(* Logix 5000 project; controller reports 1756-L63 rev 20.15; software revision 20.04; part 43 of 52 *)

        [112].log_data[48].valid := 1, [112].log_data[49].min := 6.5370584, [112].log_data[49].max := 9.345203, [112].log_data[49].total := 30173.871, [112].log_data[49].time := 3600.0, [112].log_data[49].minminute := 59, [112].log_data[49].maxminute := 34, [112].log_data[49].valid := 1, [112].log_data[50].min := 1.828552, [112].log_data[50].max := 1.9386716, [112].log_data[50].total := 6771.5327, [112].log_data[50].time := 3600.0, [112].log_data[50].minminute := 33, [112].log_data[50].maxminute := 40, [112].log_data[50].valid := 1, [112].log_data[51].time := 3600.0, [112].log_data[51].valid := 1, [112].log_data[52].min := -2.7799988, [112].log_data[52].max := 0.11999512, [112].log_data[52].total := -7734.9287, [112].log_data[52].time := 3600.0, [112].log_data[52].minminute := 1, [112].log_data[52].valid := 1, [112].log_data[53].min := -2.7000046, [112].log_data[53].max := 0.13999939, [112].log_data[53].total := -7364.768, [112].log_data[53].time := 3600.0, [112].log_data[53].minminute := 38, [112].log_data[53].maxminute := 27, [112].log_data[53].valid := 1, [112].log_data[54].max := 0.537, [112].log_data[54].total := 1216.9052, [112].log_data[54].time := 3600.0, [112].log_data[54].maxminute := 12, [112].log_data[54].valid := 1, [112].log_data[55].max := 0.528, [112].log_data[55].total := 1217.3307, [112].log_data[55].time := 3600.0, [112].log_data[55].minminute := 5, [112].log_data[55].maxminute := 38, [112].log_data[55].valid := 1, [112].log_data[56].min := 0.15938194, [112].log_data[56].max := 0.15989229, [112].log_data[56].total := 574.438, [112].log_data[56].time := 3600.0, [112].log_data[56].minminute := 2, [112].log_data[56].maxminute := 17, [112].log_data[56].valid := 1, [112].log_data[57].min := 0.22258775, [112].log_data[57].max := 0.22325513, [112].log_data[57].total := 802.80646, [112].log_data[57].time := 3600.0, [112].log_data[57].minminute := 59, [112].log_data[57].maxminute := 9, [112].log_data[57].valid := 1, [112].log_data[58].time := 3600.0, [112].log_data[58].valid := 1, [112].log_data[59].time := 3600.0, [112].log_data[59].valid := 1, [112].log_data[60].valid := 1,
        [112].log_data[61].valid := 1, [112].log_data[62].valid := 1, [112].log_data[63].valid := 1, [112].log_data[64].valid := 1, [112].log_data[65].valid := 1, [112].log_data[66].valid := 1, [112].log_data[67].valid := 1, [112].log_data[68].valid := 1, [112].log_data[69].valid := 1, [112].log_data[70].valid := 1, [112].log_data[71].valid := 1, [112].log_data[72].valid := 1, [112].log_data[73].valid := 1, [112].log_data[74].valid := 1, [112].log_data[75].valid := 1, [112].log_data[76].valid := 1, [112].log_data[77].valid := 1, [112].log_data[78].valid := 1, [112].log_data[79].valid := 1, [112].log_data[80].valid := 1, [112].log_data[81].valid := 1, [112].log_data[82].valid := 1, [112].log_data[83].valid := 1, [112].log_data[84].valid := 1, [112].log_data[85].valid := 1, [112].log_data[86].valid := 1, [112].log_data[87].valid := 1, [112].log_data[88].valid := 1, [112].log_data[89].valid := 1, [112].log_data[90].valid := 1, [112].log_data[91].valid := 1, [112].log_data[92].valid := 1, [112].log_data[93].valid := 1, [112].log_data[94].valid := 1, [112].log_data[95].valid := 1, [112].log_data[96].valid := 1, [112].log_data[97].valid := 1, [112].log_data[98].valid := 1, [112].log_data[99].valid := 1, [112].log_data[100].valid := 1, [112].log_data[101].valid := 1, [112].log_data[102].valid := 1, [112].log_data[103].valid := 1, [112].log_data[104].valid := 1, [112].log_data[105].valid := 1, [112].log_data[106].valid := 1, [112].log_data[107].valid := 1, [112].log_data[108].valid := 1, [112].log_data[109].valid := 1, [112].log_data[110].valid := 1, [112].log_data[111].valid := 1, [112].log_data[112].valid := 1, [112].log_data[113].valid := 1, [112].log_data[114].valid := 1, [112].log_data[115].valid := 1, [112].log_data[116].valid := 1, [112].log_data[117].valid := 1, [112].log_data[118].valid := 1, [112].log_data[119].valid := 1, [112].log_data[120].valid := 1,
        [112].log_data[121].valid := 1, [112].log_data[122].valid := 1, [112].log_data[123].valid := 1, [112].log_data[124].valid := 1, [112].time.Year := 2023, [112].time.Month := 1, [112].time.Day := 17, [112].time.Hour := 19, [112].time.Minute := 59, [112].time.Second := 59, [113].log_data[0].min := 1.0, [113].log_data[0].max := 1.0, [113].log_data[0].total := 3599.5, [113].log_data[0].time := 3599.5, [113].log_data[0].valid := 1, [113].log_data[1].max := 1.0, [113].log_data[1].total := 584.0, [113].log_data[1].time := 3599.5, [113].log_data[1].maxminute := 41, [113].log_data[1].valid := 1, [113].log_data[2].max := 1.0, [113].log_data[2].total := 580.5, [113].log_data[2].time := 3599.5, [113].log_data[2].maxminute := 41, [113].log_data[2].valid := 1, [113].log_data[3].time := 3599.5, [113].log_data[3].valid := 1, [113].log_data[4].time := 3599.5, [113].log_data[4].valid := 1, [113].log_data[5].max := 1.0, [113].log_data[5].total := 240.0, [113].log_data[5].time := 3599.5, [113].log_data[5].maxminute := 44, [113].log_data[5].valid := 1, [113].log_data[6].time := 3599.5, [113].log_data[6].valid := 1, [113].log_data[7].time := 3599.5, [113].log_data[7].valid := 1, [113].log_data[8].min := 1.0, [113].log_data[8].max := 1.0, [113].log_data[8].total := 3599.5, [113].log_data[8].time := 3599.5, [113].log_data[8].valid := 1, [113].log_data[9].min := 1.0, [113].log_data[9].max := 1.0, [113].log_data[9].total := 3599.5, [113].log_data[9].time := 3599.5, [113].log_data[9].valid := 1, [113].log_data[10].min := 1.0, [113].log_data[10].max := 1.0, [113].log_data[10].total := 3599.5, [113].log_data[10].time := 3599.5, [113].log_data[10].valid := 1, [113].log_data[11].time := 3599.5, [113].log_data[11].valid := 1, [113].log_data[12].min := 1.0, [113].log_data[12].max := 1.0, [113].log_data[12].total := 3599.5, [113].log_data[12].time := 3599.5, [113].log_data[12].valid := 1,
        [113].log_data[13].min := 1.0, [113].log_data[13].max := 1.0, [113].log_data[13].total := 3599.5, [113].log_data[13].time := 3599.5, [113].log_data[13].valid := 1, [113].log_data[14].time := 3599.5, [113].log_data[14].valid := 1, [113].log_data[15].time := 3599.5, [113].log_data[15].valid := 1, [113].log_data[16].time := 3599.5, [113].log_data[16].valid := 1, [113].log_data[17].min := 1.0, [113].log_data[17].max := 1.0, [113].log_data[17].total := 3599.5, [113].log_data[17].time := 3599.5, [113].log_data[17].valid := 1, [113].log_data[18].time := 3599.5, [113].log_data[18].valid := 1, [113].log_data[19].time := 3599.5, [113].log_data[19].valid := 1, [113].log_data[20].time := 3599.5, [113].log_data[20].valid := 1, [113].log_data[21].min := 1.0, [113].log_data[21].max := 1.0, [113].log_data[21].total := 3599.5, [113].log_data[21].time := 3599.5, [113].log_data[21].valid := 1, [113].log_data[22].time := 3599.5, [113].log_data[22].valid := 1, [113].log_data[23].time := 3599.5, [113].log_data[23].valid := 1, [113].log_data[24].time := 3599.5, [113].log_data[24].valid := 1, [113].log_data[25].time := 3599.5, [113].log_data[25].valid := 1, [113].log_data[26].time := 3599.5, [113].log_data[26].valid := 1, [113].log_data[27].time := 3599.5, [113].log_data[27].valid := 1, [113].log_data[28].time := 3599.5, [113].log_data[28].valid := 1, [113].log_data[29].min := 1.0, [113].log_data[29].max := 1.0, [113].log_data[29].total := 3599.5, [113].log_data[29].time := 3599.5, [113].log_data[29].valid := 1, [113].log_data[30].min := 1.0, [113].log_data[30].max := 1.0, [113].log_data[30].total := 3599.5, [113].log_data[30].time := 3599.5, [113].log_data[30].valid := 1, [113].log_data[31].max := 1.0, [113].log_data[31].total := 1629.998, [113].log_data[31].time := 3599.5, [113].log_data[31].maxminute := 4, [113].log_data[31].valid := 1, [113].log_data[32].max := 1.0, [113].log_data[32].total := 1440.749, [113].log_data[32].time := 3599.5, [113].log_data[32].minminute := 3,
        [113].log_data[32].valid := 1, [113].log_data[33].time := 3599.5, [113].log_data[33].valid := 1, [113].log_data[34].time := 3599.5, [113].log_data[34].valid := 1, [113].log_data[35].max := 1.0, [113].log_data[35].total := 1612.998, [113].log_data[35].time := 3599.5, [113].log_data[35].minminute := 8, [113].log_data[35].valid := 1, [113].log_data[36].max := 1.0, [113].log_data[36].total := 1545.498, [113].log_data[36].time := 3599.5, [113].log_data[36].maxminute := 10, [113].log_data[36].valid := 1, [113].log_data[37].max := 7.248582, [113].log_data[37].total := 3680.7366, [113].log_data[37].time := 3599.5, [113].log_data[37].maxminute := 42, [113].log_data[37].valid := 1, [113].log_data[38].time := 3599.5, [113].log_data[38].valid := 1, [113].log_data[39].min := 0.99529505, [113].log_data[39].max := 1.0213233, [113].log_data[39].total := 3605.5806, [113].log_data[39].time := 3599.5, [113].log_data[39].minminute := 13, [113].log_data[39].maxminute := 48, [113].log_data[39].valid := 1, [113].log_data[40].min := 7.6000414, [113].log_data[40].max := 7.6104846, [113].log_data[40].total := 27370.186, [113].log_data[40].time := 3599.5, [113].log_data[40].maxminute := 5, [113].log_data[40].valid := 1, [113].log_data[41].min := 0.02273633, [113].log_data[41].max := 0.023128908, [113].log_data[41].total := 82.56649, [113].log_data[41].time := 3599.5, [113].log_data[41].valid := 1, [113].log_data[42].min := 2.2916427, [113].log_data[42].max := 2.296236, [113].log_data[42].total := 8257.852, [113].log_data[42].time := 3599.5, [113].log_data[42].minminute := 53, [113].log_data[42].maxminute := 15, [113].log_data[42].valid := 1, [113].log_data[43].min := -0.27999878, [113].log_data[43].max := -0.26000214, [113].log_data[43].total := -937.77563, [113].log_data[43].time := 3599.5, [113].log_data[43].minminute := 1, [113].log_data[43].valid := 1, [113].log_data[44].min := -0.30000305, [113].log_data[44].max := -0.27999878, [113].log_data[44].total := -1079.936, [113].log_data[44].time := 3599.5, [113].log_data[44].maxminute := 50, [113].log_data[44].valid := 1, [113].log_data[45].time := 3599.5,
        [113].log_data[45].valid := 1, [113].log_data[46].time := 3599.5, [113].log_data[46].valid := 1, [113].log_data[47].time := 3599.5, [113].log_data[47].valid := 1, [113].log_data[48].min := 6.5725355, [113].log_data[48].max := 6.9006553, [113].log_data[48].total := 24290.994, [113].log_data[48].time := 3599.5, [113].log_data[48].minminute := 2, [113].log_data[48].maxminute := 51, [113].log_data[48].valid := 1, [113].log_data[49].min := 6.545106, [113].log_data[49].max := 9.279053, [113].log_data[49].total := 29584.62, [113].log_data[49].time := 3599.5, [113].log_data[49].maxminute := 44, [113].log_data[49].valid := 1, [113].log_data[50].min := 1.8549335, [113].log_data[50].max := 1.9629332, [113].log_data[50].total := 6841.0234, [113].log_data[50].time := 3599.5, [113].log_data[50].minminute := 44, [113].log_data[50].maxminute := 51, [113].log_data[50].valid := 1, [113].log_data[51].time := 3599.5, [113].log_data[51].valid := 1, [113].log_data[52].min := -2.9400024, [113].log_data[52].max := 0.11999512, [113].log_data[52].total := -7727.33, [113].log_data[52].time := 3599.5, [113].log_data[52].minminute := 4, [113].log_data[52].maxminute := 3, [113].log_data[52].valid := 1, [113].log_data[53].min := -2.540001, [113].log_data[53].max := 0.19999695, [113].log_data[53].total := -7567.941, [113].log_data[53].time := 3599.5, [113].log_data[53].minminute := 5, [113].log_data[53].maxminute := 9, [113].log_data[53].valid := 1, [113].log_data[54].max := 0.5625, [113].log_data[54].total := 1217.5094, [113].log_data[54].time := 3599.5, [113].log_data[54].minminute := 3, [113].log_data[54].maxminute := 4, [113].log_data[54].valid := 1, [113].log_data[55].max := 0.5285, [113].log_data[55].total := 1254.1487, [113].log_data[55].time := 3599.5, [113].log_data[55].minminute := 8, [113].log_data[55].maxminute := 41, [113].log_data[55].valid := 1, [113].log_data[56].min := 0.15934268, [113].log_data[56].max := 0.15985303, [113].log_data[56].total := 574.3513, [113].log_data[56].time := 3599.5, [113].log_data[56].minminute := 14, [113].log_data[56].maxminute := 17, [113].log_data[56].valid := 1,
        [113].log_data[57].min := 0.22109595, [113].log_data[57].max := 0.22278403, [113].log_data[57].total := 796.9579, [113].log_data[57].time := 3599.5, [113].log_data[57].minminute := 33, [113].log_data[57].valid := 1, [113].log_data[58].time := 3599.5, [113].log_data[58].valid := 1, [113].log_data[59].time := 3599.5, [113].log_data[59].valid := 1, [113].log_data[60].valid := 1, [113].log_data[61].valid := 1, [113].log_data[62].valid := 1, [113].log_data[63].valid := 1, [113].log_data[64].valid := 1, [113].log_data[65].valid := 1, [113].log_data[66].valid := 1, [113].log_data[67].valid := 1, [113].log_data[68].valid := 1, [113].log_data[69].valid := 1, [113].log_data[70].valid := 1, [113].log_data[71].valid := 1, [113].log_data[72].valid := 1, [113].log_data[73].valid := 1, [113].log_data[74].valid := 1, [113].log_data[75].valid := 1, [113].log_data[76].valid := 1, [113].log_data[77].valid := 1, [113].log_data[78].valid := 1, [113].log_data[79].valid := 1, [113].log_data[80].valid := 1, [113].log_data[81].valid := 1, [113].log_data[82].valid := 1, [113].log_data[83].valid := 1, [113].log_data[84].valid := 1, [113].log_data[85].valid := 1, [113].log_data[86].valid := 1, [113].log_data[87].valid := 1, [113].log_data[88].valid := 1, [113].log_data[89].valid := 1, [113].log_data[90].valid := 1, [113].log_data[91].valid := 1, [113].log_data[92].valid := 1, [113].log_data[93].valid := 1, [113].log_data[94].valid := 1, [113].log_data[95].valid := 1, [113].log_data[96].valid := 1, [113].log_data[97].valid := 1, [113].log_data[98].valid := 1, [113].log_data[99].valid := 1, [113].log_data[100].valid := 1, [113].log_data[101].valid := 1, [113].log_data[102].valid := 1, [113].log_data[103].valid := 1, [113].log_data[104].valid := 1, [113].log_data[105].valid := 1, [113].log_data[106].valid := 1, [113].log_data[107].valid := 1, [113].log_data[108].valid := 1, [113].log_data[109].valid := 1,
        [113].log_data[110].valid := 1, [113].log_data[111].valid := 1, [113].log_data[112].valid := 1, [113].log_data[113].valid := 1, [113].log_data[114].valid := 1, [113].log_data[115].valid := 1, [113].log_data[116].valid := 1, [113].log_data[117].valid := 1, [113].log_data[118].valid := 1, [113].log_data[119].valid := 1, [113].log_data[120].valid := 1, [113].log_data[121].valid := 1, [113].log_data[122].valid := 1, [113].log_data[123].valid := 1, [113].log_data[124].valid := 1, [113].time.Year := 2023, [113].time.Month := 1, [113].time.Day := 17, [113].time.Hour := 20, [113].time.Minute := 59, [113].time.Second := 59, [114].log_data[0].min := 1.0, [114].log_data[0].max := 1.0, [114].log_data[0].total := 3600.0, [114].log_data[0].time := 3600.0, [114].log_data[0].valid := 1, [114].log_data[1].max := 1.0, [114].log_data[1].total := 555.5, [114].log_data[1].time := 3600.0, [114].log_data[1].maxminute := 46, [114].log_data[1].valid := 1, [114].log_data[2].max := 1.0, [114].log_data[2].total := 552.0, [114].log_data[2].time := 3600.0, [114].log_data[2].maxminute := 46, [114].log_data[2].valid := 1, [114].log_data[3].time := 3600.0, [114].log_data[3].valid := 1, [114].log_data[4].time := 3600.0, [114].log_data[4].valid := 1, [114].log_data[5].max := 1.0, [114].log_data[5].total := 244.0, [114].log_data[5].time := 3600.0, [114].log_data[5].maxminute := 49, [114].log_data[5].valid := 1, [114].log_data[6].time := 3600.0, [114].log_data[6].valid := 1, [114].log_data[7].time := 3600.0, [114].log_data[7].valid := 1, [114].log_data[8].min := 1.0, [114].log_data[8].max := 1.0, [114].log_data[8].total := 3600.0, [114].log_data[8].time := 3600.0, [114].log_data[8].valid := 1, [114].log_data[9].min := 1.0, [114].log_data[9].max := 1.0, [114].log_data[9].total := 3600.0, [114].log_data[9].time := 3600.0, [114].log_data[9].valid := 1, [114].log_data[10].min := 1.0,
        [114].log_data[10].max := 1.0, [114].log_data[10].total := 3600.0, [114].log_data[10].time := 3600.0, [114].log_data[10].valid := 1, [114].log_data[11].time := 3600.0, [114].log_data[11].valid := 1, [114].log_data[12].min := 1.0, [114].log_data[12].max := 1.0, [114].log_data[12].total := 3600.0, [114].log_data[12].time := 3600.0, [114].log_data[12].valid := 1, [114].log_data[13].min := 1.0, [114].log_data[13].max := 1.0, [114].log_data[13].total := 3600.0, [114].log_data[13].time := 3600.0, [114].log_data[13].valid := 1, [114].log_data[14].time := 3600.0, [114].log_data[14].valid := 1, [114].log_data[15].time := 3600.0, [114].log_data[15].valid := 1, [114].log_data[16].time := 3600.0, [114].log_data[16].valid := 1, [114].log_data[17].min := 1.0, [114].log_data[17].max := 1.0, [114].log_data[17].total := 3600.0, [114].log_data[17].time := 3600.0, [114].log_data[17].valid := 1, [114].log_data[18].time := 3600.0, [114].log_data[18].valid := 1, [114].log_data[19].time := 3600.0, [114].log_data[19].valid := 1, [114].log_data[20].time := 3600.0, [114].log_data[20].valid := 1, [114].log_data[21].min := 1.0, [114].log_data[21].max := 1.0, [114].log_data[21].total := 3600.0, [114].log_data[21].time := 3600.0, [114].log_data[21].valid := 1, [114].log_data[22].time := 3600.0, [114].log_data[22].valid := 1, [114].log_data[23].time := 3600.0, [114].log_data[23].valid := 1, [114].log_data[24].time := 3600.0, [114].log_data[24].valid := 1, [114].log_data[25].time := 3600.0, [114].log_data[25].valid := 1, [114].log_data[26].time := 3600.0, [114].log_data[26].valid := 1, [114].log_data[27].time := 3600.0, [114].log_data[27].valid := 1, [114].log_data[28].time := 3600.0, [114].log_data[28].valid := 1, [114].log_data[29].min := 1.0, [114].log_data[29].max := 1.0, [114].log_data[29].total := 3600.0, [114].log_data[29].time := 3600.0, [114].log_data[29].valid := 1, [114].log_data[30].min := 1.0, [114].log_data[30].max := 1.0, [114].log_data[30].total := 3600.0,
        [114].log_data[30].time := 3600.0, [114].log_data[30].valid := 1, [114].log_data[31].max := 1.0, [114].log_data[31].total := 1629.7471, [114].log_data[31].time := 3600.0, [114].log_data[31].maxminute := 7, [114].log_data[31].valid := 1, [114].log_data[32].max := 1.0, [114].log_data[32].total := 1466.749, [114].log_data[32].time := 3600.0, [114].log_data[32].minminute := 6, [114].log_data[32].valid := 1, [114].log_data[33].time := 3600.0, [114].log_data[33].valid := 1, [114].log_data[34].time := 3600.0, [114].log_data[34].valid := 1, [114].log_data[35].max := 1.0, [114].log_data[35].total := 1629.998, [114].log_data[35].time := 3600.0, [114].log_data[35].maxminute := 2, [114].log_data[35].valid := 1, [114].log_data[36].max := 1.0, [114].log_data[36].total := 1440.7471, [114].log_data[36].time := 3600.0, [114].log_data[36].minminute := 1, [114].log_data[36].valid := 1, [114].log_data[37].max := 7.5233893, [114].log_data[37].total := 3622.97, [114].log_data[37].time := 3600.0, [114].log_data[37].maxminute := 47, [114].log_data[37].valid := 1, [114].log_data[38].time := 3600.0, [114].log_data[38].valid := 1, [114].log_data[39].min := 0.9960017, [114].log_data[39].max := 1.0210879, [114].log_data[39].total := 3610.188, [114].log_data[39].time := 3600.0, [114].log_data[39].minminute := 34, [114].log_data[39].maxminute := 49, [114].log_data[39].valid := 1, [114].log_data[40].min := 7.5885, [114].log_data[40].max := 7.611859, [114].log_data[40].total := 27368.842, [114].log_data[40].time := 3600.0, [114].log_data[40].minminute := 14, [114].log_data[40].maxminute := 25, [114].log_data[40].valid := 1, [114].log_data[41].min := 0.02273633, [114].log_data[41].max := 0.023128908, [114].log_data[41].total := 82.563736, [114].log_data[41].time := 3600.0, [114].log_data[41].valid := 1, [114].log_data[42].min := 2.2917604, [114].log_data[42].max := 2.296236, [114].log_data[42].total := 8259.057, [114].log_data[42].time := 3600.0, [114].log_data[42].minminute := 39, [114].log_data[42].maxminute := 24, [114].log_data[42].valid := 1, [114].log_data[43].min := -0.27999878,
        [114].log_data[43].max := -0.26000214, [114].log_data[43].total := -938.5357, [114].log_data[43].time := 3600.0, [114].log_data[43].valid := 1, [114].log_data[44].min := -0.30000305, [114].log_data[44].max := -0.27999878, [114].log_data[44].total := -1080.0408, [114].log_data[44].time := 3600.0, [114].log_data[44].valid := 1, [114].log_data[45].time := 3600.0, [114].log_data[45].valid := 1, [114].log_data[46].time := 3600.0, [114].log_data[46].valid := 1, [114].log_data[47].time := 3600.0, [114].log_data[47].valid := 1, [114].log_data[48].min := 6.578031, [114].log_data[48].max := 6.9179688, [114].log_data[48].total := 24247.959, [114].log_data[48].time := 3600.0, [114].log_data[48].minminute := 13, [114].log_data[48].maxminute := 56, [114].log_data[48].valid := 1, [114].log_data[49].min := 6.600068, [114].log_data[49].max := 9.21408, [114].log_data[49].total := 28705.174, [114].log_data[49].time := 3600.0, [114].log_data[49].minminute := 9, [114].log_data[49].maxminute := 49, [114].log_data[49].valid := 1, [114].log_data[50].min := 1.8884994, [114].log_data[50].max := 1.9981477, [114].log_data[50].total := 6944.73, [114].log_data[50].time := 3600.0, [114].log_data[50].minminute := 49, [114].log_data[50].maxminute := 55, [114].log_data[50].valid := 1, [114].log_data[51].time := 3600.0, [114].log_data[51].valid := 1, [114].log_data[52].min := -3.0, [114].log_data[52].max := 0.11999512, [114].log_data[52].total := -7840.5713, [114].log_data[52].time := 3600.0, [114].log_data[52].minminute := 28, [114].log_data[52].maxminute := 6, [114].log_data[52].valid := 1, [114].log_data[53].min := -2.5600052, [114].log_data[53].max := 0.11999512, [114].log_data[53].total := -7368.902, [114].log_data[53].time := 3600.0, [114].log_data[53].minminute := 34, [114].log_data[53].maxminute := 2, [114].log_data[53].valid := 1, [114].log_data[54].max := 0.549, [114].log_data[54].total := 1229.9313, [114].log_data[54].time := 3600.0, [114].log_data[54].minminute := 6, [114].log_data[54].maxminute := 28, [114].log_data[54].valid := 1, [114].log_data[55].max := 0.53, [114].log_data[55].total := 1217.2065,
        [114].log_data[55].time := 3600.0, [114].log_data[55].minminute := 1, [114].log_data[55].maxminute := 34, [114].log_data[55].valid := 1, [114].log_data[56].min := 0.15934268, [114].log_data[56].max := 0.15989229, [114].log_data[56].total := 574.4744, [114].log_data[56].time := 3600.0, [114].log_data[56].minminute := 6, [114].log_data[56].maxminute := 20, [114].log_data[56].valid := 1, [114].log_data[57].min := 0.21964341, [114].log_data[57].max := 0.22148852, [114].log_data[57].total := 792.6085, [114].log_data[57].time := 3600.0, [114].log_data[57].minminute := 37, [114].log_data[57].valid := 1, [114].log_data[58].time := 3600.0, [114].log_data[58].valid := 1, [114].log_data[59].time := 3600.0, [114].log_data[59].valid := 1, [114].log_data[60].valid := 1, [114].log_data[61].valid := 1, [114].log_data[62].valid := 1, [114].log_data[63].valid := 1, [114].log_data[64].valid := 1, [114].log_data[65].valid := 1, [114].log_data[66].valid := 1, [114].log_data[67].valid := 1, [114].log_data[68].valid := 1, [114].log_data[69].valid := 1, [114].log_data[70].valid := 1, [114].log_data[71].valid := 1, [114].log_data[72].valid := 1, [114].log_data[73].valid := 1, [114].log_data[74].valid := 1, [114].log_data[75].valid := 1, [114].log_data[76].valid := 1, [114].log_data[77].valid := 1, [114].log_data[78].valid := 1, [114].log_data[79].valid := 1, [114].log_data[80].valid := 1, [114].log_data[81].valid := 1, [114].log_data[82].valid := 1, [114].log_data[83].valid := 1, [114].log_data[84].valid := 1, [114].log_data[85].valid := 1, [114].log_data[86].valid := 1, [114].log_data[87].valid := 1, [114].log_data[88].valid := 1, [114].log_data[89].valid := 1, [114].log_data[90].valid := 1, [114].log_data[91].valid := 1, [114].log_data[92].valid := 1, [114].log_data[93].valid := 1, [114].log_data[94].valid := 1, [114].log_data[95].valid := 1, [114].log_data[96].valid := 1, [114].log_data[97].valid := 1, [114].log_data[98].valid := 1,
        [114].log_data[99].valid := 1, [114].log_data[100].valid := 1, [114].log_data[101].valid := 1, [114].log_data[102].valid := 1, [114].log_data[103].valid := 1, [114].log_data[104].valid := 1, [114].log_data[105].valid := 1, [114].log_data[106].valid := 1, [114].log_data[107].valid := 1, [114].log_data[108].valid := 1, [114].log_data[109].valid := 1, [114].log_data[110].valid := 1, [114].log_data[111].valid := 1, [114].log_data[112].valid := 1, [114].log_data[113].valid := 1, [114].log_data[114].valid := 1, [114].log_data[115].valid := 1, [114].log_data[116].valid := 1, [114].log_data[117].valid := 1, [114].log_data[118].valid := 1, [114].log_data[119].valid := 1, [114].log_data[120].valid := 1, [114].log_data[121].valid := 1, [114].log_data[122].valid := 1, [114].log_data[123].valid := 1, [114].log_data[124].valid := 1, [114].time.Year := 2023, [114].time.Month := 1, [114].time.Day := 17, [114].time.Hour := 21, [114].time.Minute := 59, [114].time.Second := 59, [115].log_data[0].min := 1.0, [115].log_data[0].max := 1.0, [115].log_data[0].total := 3600.0, [115].log_data[0].time := 3600.0, [115].log_data[0].valid := 1, [115].log_data[1].time := 3600.0, [115].log_data[1].valid := 1, [115].log_data[2].time := 3600.0, [115].log_data[2].valid := 1, [115].log_data[3].time := 3600.0, [115].log_data[3].valid := 1, [115].log_data[4].time := 3600.0, [115].log_data[4].valid := 1, [115].log_data[5].time := 3600.0, [115].log_data[5].valid := 1, [115].log_data[6].time := 3600.0, [115].log_data[6].valid := 1, [115].log_data[7].time := 3600.0, [115].log_data[7].valid := 1, [115].log_data[8].min := 1.0, [115].log_data[8].max := 1.0, [115].log_data[8].total := 3600.0, [115].log_data[8].time := 3600.0, [115].log_data[8].valid := 1, [115].log_data[9].min := 1.0, [115].log_data[9].max := 1.0, [115].log_data[9].total := 3600.0, [115].log_data[9].time := 3600.0,
        [115].log_data[9].valid := 1, [115].log_data[10].min := 1.0, [115].log_data[10].max := 1.0, [115].log_data[10].total := 3600.0, [115].log_data[10].time := 3600.0, [115].log_data[10].valid := 1, [115].log_data[11].time := 3600.0, [115].log_data[11].valid := 1, [115].log_data[12].min := 1.0, [115].log_data[12].max := 1.0, [115].log_data[12].total := 3600.0, [115].log_data[12].time := 3600.0, [115].log_data[12].valid := 1, [115].log_data[13].min := 1.0, [115].log_data[13].max := 1.0, [115].log_data[13].total := 3600.0, [115].log_data[13].time := 3600.0, [115].log_data[13].valid := 1, [115].log_data[14].time := 3600.0, [115].log_data[14].valid := 1, [115].log_data[15].time := 3600.0, [115].log_data[15].valid := 1, [115].log_data[16].time := 3600.0, [115].log_data[16].valid := 1, [115].log_data[17].min := 1.0, [115].log_data[17].max := 1.0, [115].log_data[17].total := 3600.0, [115].log_data[17].time := 3600.0, [115].log_data[17].valid := 1, [115].log_data[18].time := 3600.0, [115].log_data[18].valid := 1, [115].log_data[19].time := 3600.0, [115].log_data[19].valid := 1, [115].log_data[20].time := 3600.0, [115].log_data[20].valid := 1, [115].log_data[21].min := 1.0, [115].log_data[21].max := 1.0, [115].log_data[21].total := 3600.0, [115].log_data[21].time := 3600.0, [115].log_data[21].valid := 1, [115].log_data[22].time := 3600.0, [115].log_data[22].valid := 1, [115].log_data[23].time := 3600.0, [115].log_data[23].valid := 1, [115].log_data[24].time := 3600.0, [115].log_data[24].valid := 1, [115].log_data[25].time := 3600.0, [115].log_data[25].valid := 1, [115].log_data[26].time := 3600.0, [115].log_data[26].valid := 1, [115].log_data[27].time := 3600.0, [115].log_data[27].valid := 1, [115].log_data[28].time := 3600.0, [115].log_data[28].valid := 1, [115].log_data[29].min := 1.0, [115].log_data[29].max := 1.0, [115].log_data[29].total := 3600.0, [115].log_data[29].time := 3600.0, [115].log_data[29].valid := 1, [115].log_data[30].min := 1.0,
        [115].log_data[30].max := 1.0, [115].log_data[30].total := 3600.0, [115].log_data[30].time := 3600.0, [115].log_data[30].valid := 1, [115].log_data[31].max := 1.0, [115].log_data[31].total := 1503.2471, [115].log_data[31].time := 3600.0, [115].log_data[31].maxminute := 10, [115].log_data[31].valid := 1, [115].log_data[32].max := 1.0, [115].log_data[32].total := 1629.7471, [115].log_data[32].time := 3600.0, [115].log_data[32].valid := 1, [115].log_data[33].time := 3600.0, [115].log_data[33].valid := 1, [115].log_data[34].time := 3600.0, [115].log_data[34].valid := 1, [115].log_data[35].max := 1.0, [115].log_data[35].total := 1629.7471, [115].log_data[35].time := 3600.0, [115].log_data[35].maxminute := 6, [115].log_data[35].valid := 1, [115].log_data[36].max := 1.0, [115].log_data[36].total := 1440.7471, [115].log_data[36].time := 3600.0, [115].log_data[36].minminute := 4, [115].log_data[36].valid := 1, [115].log_data[37].time := 3600.0, [115].log_data[37].valid := 1, [115].log_data[38].time := 3600.0, [115].log_data[38].valid := 1, [115].log_data[39].min := 0.99635506, [115].log_data[39].max := 1.0057771, [115].log_data[39].total := 3606.2104, [115].log_data[39].time := 3600.0, [115].log_data[39].minminute := 50, [115].log_data[39].maxminute := 38, [115].log_data[39].valid := 1, [115].log_data[40].min := 7.5959196, [115].log_data[40].max := 7.6093855, [115].log_data[40].total := 27370.8, [115].log_data[40].time := 3600.0, [115].log_data[40].minminute := 51, [115].log_data[40].maxminute := 44, [115].log_data[40].valid := 1, [115].log_data[41].min := 0.02273633, [115].log_data[41].max := 0.023128908, [115].log_data[41].total := 82.562836, [115].log_data[41].time := 3600.0, [115].log_data[41].valid := 1, [115].log_data[42].min := 2.291525, [115].log_data[42].max := 2.296118, [115].log_data[42].total := 8258.939, [115].log_data[42].time := 3600.0, [115].log_data[42].minminute := 48, [115].log_data[42].maxminute := 43, [115].log_data[42].valid := 1, [115].log_data[43].min := -0.27999878, [115].log_data[43].max := -0.26000214, [115].log_data[43].total := -942.2139,
        [115].log_data[43].time := 3600.0, [115].log_data[43].valid := 1, [115].log_data[44].min := -0.30000305, [115].log_data[44].max := -0.27999878, [115].log_data[44].total := -1080.086, [115].log_data[44].time := 3600.0, [115].log_data[44].maxminute := 7, [115].log_data[44].valid := 1, [115].log_data[45].time := 3600.0, [115].log_data[45].valid := 1, [115].log_data[46].time := 3600.0, [115].log_data[46].valid := 1, [115].log_data[47].time := 3600.0, [115].log_data[47].valid := 1, [115].log_data[48].min := 6.5810537, [115].log_data[48].max := 6.7981515, [115].log_data[48].total := 24189.363, [115].log_data[48].time := 3600.0, [115].log_data[48].minminute := 19, [115].log_data[48].maxminute := 34, [115].log_data[48].valid := 1, [115].log_data[49].min := 6.5562954, [115].log_data[49].max := 9.285334, [115].log_data[49].total := 28568.717, [115].log_data[49].time := 3600.0, [115].log_data[49].minminute := 15, [115].log_data[49].maxminute := 59, [115].log_data[49].valid := 1, [115].log_data[50].min := 1.913821, [115].log_data[50].max := 1.9932013, [115].log_data[50].total := 7037.052, [115].log_data[50].time := 3600.0, [115].log_data[50].minminute := 58, [115].log_data[50].valid := 1, [115].log_data[51].time := 3600.0, [115].log_data[51].valid := 1, [115].log_data[52].min := -2.7600021, [115].log_data[52].max := 0.11999512, [115].log_data[52].total := -7917.2695, [115].log_data[52].time := 3600.0, [115].log_data[52].minminute := 32, [115].log_data[52].valid := 1, [115].log_data[53].min := -2.540001, [115].log_data[53].max := 0.27999878, [115].log_data[53].total := -7346.545, [115].log_data[53].time := 3600.0, [115].log_data[53].minminute := 35, [115].log_data[53].maxminute := 26, [115].log_data[53].valid := 1, [115].log_data[54].max := 0.517, [115].log_data[54].total := 1241.6158, [115].log_data[54].time := 3600.0, [115].log_data[54].maxminute := 53, [115].log_data[54].valid := 1, [115].log_data[55].max := 0.5545, [115].log_data[55].total := 1217.3616, [115].log_data[55].time := 3600.0, [115].log_data[55].minminute := 4, [115].log_data[55].maxminute := 48, [115].log_data[55].valid := 1,
        [115].log_data[56].min := 0.15930341, [115].log_data[56].max := 0.15981378, [115].log_data[56].total := 574.40155, [115].log_data[56].time := 3600.0, [115].log_data[56].minminute := 14, [115].log_data[56].maxminute := 14, [115].log_data[56].valid := 1, [115].log_data[57].min := 0.21803379, [115].log_data[57].max := 0.21995747, [115].log_data[57].total := 787.6007, [115].log_data[57].time := 3600.0, [115].log_data[57].minminute := 58, [115].log_data[57].valid := 1, [115].log_data[58].time := 3600.0, [115].log_data[58].valid := 1, [115].log_data[59].time := 3600.0, [115].log_data[59].valid := 1, [115].log_data[60].valid := 1, [115].log_data[61].valid := 1, [115].log_data[62].valid := 1, [115].log_data[63].valid := 1, [115].log_data[64].valid := 1, [115].log_data[65].valid := 1, [115].log_data[66].valid := 1, [115].log_data[67].valid := 1, [115].log_data[68].valid := 1, [115].log_data[69].valid := 1, [115].log_data[70].valid := 1, [115].log_data[71].valid := 1, [115].log_data[72].valid := 1, [115].log_data[73].valid := 1, [115].log_data[74].valid := 1, [115].log_data[75].valid := 1, [115].log_data[76].valid := 1, [115].log_data[77].valid := 1, [115].log_data[78].valid := 1, [115].log_data[79].valid := 1, [115].log_data[80].valid := 1, [115].log_data[81].valid := 1, [115].log_data[82].valid := 1, [115].log_data[83].valid := 1, [115].log_data[84].valid := 1, [115].log_data[85].valid := 1, [115].log_data[86].valid := 1, [115].log_data[87].valid := 1, [115].log_data[88].valid := 1, [115].log_data[89].valid := 1, [115].log_data[90].valid := 1, [115].log_data[91].valid := 1, [115].log_data[92].valid := 1, [115].log_data[93].valid := 1, [115].log_data[94].valid := 1, [115].log_data[95].valid := 1, [115].log_data[96].valid := 1, [115].log_data[97].valid := 1, [115].log_data[98].valid := 1, [115].log_data[99].valid := 1, [115].log_data[100].valid := 1, [115].log_data[101].valid := 1, [115].log_data[102].valid := 1,
        [115].log_data[103].valid := 1, [115].log_data[104].valid := 1, [115].log_data[105].valid := 1, [115].log_data[106].valid := 1, [115].log_data[107].valid := 1, [115].log_data[108].valid := 1, [115].log_data[109].valid := 1, [115].log_data[110].valid := 1, [115].log_data[111].valid := 1, [115].log_data[112].valid := 1, [115].log_data[113].valid := 1, [115].log_data[114].valid := 1, [115].log_data[115].valid := 1, [115].log_data[116].valid := 1, [115].log_data[117].valid := 1, [115].log_data[118].valid := 1, [115].log_data[119].valid := 1, [115].log_data[120].valid := 1, [115].log_data[121].valid := 1, [115].log_data[122].valid := 1, [115].log_data[123].valid := 1, [115].log_data[124].valid := 1, [115].time.Year := 2023, [115].time.Month := 1, [115].time.Day := 17, [115].time.Hour := 22, [115].time.Minute := 59, [115].time.Second := 59, [116].log_data[0].min := 1.0, [116].log_data[0].max := 1.0, [116].log_data[0].total := 3600.0, [116].log_data[0].time := 3600.0, [116].log_data[0].valid := 1, [116].log_data[1].max := 1.0, [116].log_data[1].total := 561.5, [116].log_data[1].time := 3600.0, [116].log_data[1].maxminute := 5, [116].log_data[1].valid := 1, [116].log_data[2].max := 1.0, [116].log_data[2].total := 558.0, [116].log_data[2].time := 3600.0, [116].log_data[2].maxminute := 5, [116].log_data[2].valid := 1, [116].log_data[3].time := 3600.0, [116].log_data[3].valid := 1, [116].log_data[4].time := 3600.0, [116].log_data[4].valid := 1, [116].log_data[5].max := 1.0, [116].log_data[5].total := 240.0, [116].log_data[5].time := 3600.0, [116].log_data[5].maxminute := 7, [116].log_data[5].valid := 1, [116].log_data[6].time := 3600.0, [116].log_data[6].valid := 1, [116].log_data[7].time := 3600.0, [116].log_data[7].valid := 1, [116].log_data[8].min := 1.0, [116].log_data[8].max := 1.0, [116].log_data[8].total := 3600.0, [116].log_data[8].time := 3600.0,
        [116].log_data[8].valid := 1, [116].log_data[9].min := 1.0, [116].log_data[9].max := 1.0, [116].log_data[9].total := 3600.0, [116].log_data[9].time := 3600.0, [116].log_data[9].valid := 1, [116].log_data[10].min := 1.0, [116].log_data[10].max := 1.0, [116].log_data[10].total := 3600.0, [116].log_data[10].time := 3600.0, [116].log_data[10].valid := 1, [116].log_data[11].time := 3600.0, [116].log_data[11].valid := 1, [116].log_data[12].min := 1.0, [116].log_data[12].max := 1.0, [116].log_data[12].total := 3600.0, [116].log_data[12].time := 3600.0, [116].log_data[12].valid := 1, [116].log_data[13].min := 1.0, [116].log_data[13].max := 1.0, [116].log_data[13].total := 3600.0, [116].log_data[13].time := 3600.0, [116].log_data[13].valid := 1, [116].log_data[14].time := 3600.0, [116].log_data[14].valid := 1, [116].log_data[15].time := 3600.0, [116].log_data[15].valid := 1, [116].log_data[16].time := 3600.0, [116].log_data[16].valid := 1, [116].log_data[17].min := 1.0, [116].log_data[17].max := 1.0, [116].log_data[17].total := 3600.0, [116].log_data[17].time := 3600.0, [116].log_data[17].valid := 1, [116].log_data[18].time := 3600.0, [116].log_data[18].valid := 1, [116].log_data[19].time := 3600.0, [116].log_data[19].valid := 1, [116].log_data[20].time := 3600.0, [116].log_data[20].valid := 1, [116].log_data[21].min := 1.0, [116].log_data[21].max := 1.0, [116].log_data[21].total := 3600.0, [116].log_data[21].time := 3600.0, [116].log_data[21].valid := 1, [116].log_data[22].time := 3600.0, [116].log_data[22].valid := 1, [116].log_data[23].time := 3600.0, [116].log_data[23].valid := 1, [116].log_data[24].time := 3600.0, [116].log_data[24].valid := 1, [116].log_data[25].time := 3600.0, [116].log_data[25].valid := 1, [116].log_data[26].time := 3600.0, [116].log_data[26].valid := 1, [116].log_data[27].time := 3600.0, [116].log_data[27].valid := 1, [116].log_data[28].time := 3600.0, [116].log_data[28].valid := 1, [116].log_data[29].min := 1.0,
        [116].log_data[29].max := 1.0, [116].log_data[29].total := 3600.0, [116].log_data[29].time := 3600.0, [116].log_data[29].valid := 1, [116].log_data[30].min := 1.0, [116].log_data[30].max := 1.0, [116].log_data[30].total := 3600.0, [116].log_data[30].time := 3600.0, [116].log_data[30].valid := 1, [116].log_data[31].max := 1.0, [116].log_data[31].total := 1440.7471, [116].log_data[31].time := 3600.0, [116].log_data[31].minminute := 2, [116].log_data[31].valid := 1, [116].log_data[32].max := 1.0, [116].log_data[32].total := 1629.998, [116].log_data[32].time := 3600.0, [116].log_data[32].maxminute := 3, [116].log_data[32].valid := 1, [116].log_data[33].time := 3600.0, [116].log_data[33].valid := 1, [116].log_data[34].time := 3600.0, [116].log_data[34].valid := 1, [116].log_data[35].max := 1.0, [116].log_data[35].total := 1609.7471, [116].log_data[35].time := 3600.0, [116].log_data[35].maxminute := 9, [116].log_data[35].valid := 1, [116].log_data[36].max := 1.0, [116].log_data[36].total := 1548.998, [116].log_data[36].time := 3600.0, [116].log_data[36].minminute := 7, [116].log_data[36].valid := 1, [116].log_data[37].max := 7.209323, [116].log_data[37].total := 3524.1855, [116].log_data[37].time := 3600.0, [116].log_data[37].maxminute := 5, [116].log_data[37].valid := 1, [116].log_data[38].time := 3600.0, [116].log_data[38].valid := 1, [116].log_data[39].min := 0.9956484, [116].log_data[39].max := 1.02203, [116].log_data[39].total := 3608.7498, [116].log_data[39].time := 3600.0, [116].log_data[39].minminute := 46, [116].log_data[39].maxminute := 7, [116].log_data[39].valid := 1, [116].log_data[40].min := 7.5972934, [116].log_data[40].max := 7.6104846, [116].log_data[40].total := 27377.336, [116].log_data[40].time := 3600.0, [116].log_data[40].minminute := 51, [116].log_data[40].maxminute := 54, [116].log_data[40].valid := 1, [116].log_data[41].min := 0.02273633, [116].log_data[41].max := 0.023325196, [116].log_data[41].total := 82.61728, [116].log_data[41].time := 3600.0, [116].log_data[41].maxminute := 7, [116].log_data[41].valid := 1,
        [116].log_data[42].min := 2.2916427, [116].log_data[42].max := 2.2965894, [116].log_data[42].total := 8259.007, [116].log_data[42].time := 3600.0, [116].log_data[42].minminute := 34, [116].log_data[42].maxminute := 7, [116].log_data[42].valid := 1, [116].log_data[43].min := -0.27999878, [116].log_data[43].max := -0.26000214, [116].log_data[43].total := -942.9897, [116].log_data[43].time := 3600.0, [116].log_data[43].valid := 1, [116].log_data[44].min := -0.30000305, [116].log_data[44].max := -0.30000305, [116].log_data[44].total := -1080.0911, [116].log_data[44].time := 3600.0, [116].log_data[44].valid := 1, [116].log_data[45].time := 3600.0, [116].log_data[45].valid := 1, [116].log_data[46].time := 3600.0, [116].log_data[46].valid := 1, [116].log_data[47].time := 3600.0, [116].log_data[47].valid := 1, [116].log_data[48].min := 6.5821533, [116].log_data[48].max := 6.9196177, [116].log_data[48].total := 24232.64, [116].log_data[48].time := 3600.0, [116].log_data[48].minminute := 38, [116].log_data[48].maxminute := 14, [116].log_data[48].valid := 1, [116].log_data[49].min := 6.570625, [116].log_data[49].max := 9.333033, [116].log_data[49].total := 28300.158, [116].log_data[49].time := 3600.0, [116].log_data[49].minminute := 32, [116].log_data[49].maxminute := 8, [116].log_data[49].valid := 1, [116].log_data[50].min := 1.9000413, [116].log_data[50].max := 2.0099254, [116].log_data[50].total := 7091.859, [116].log_data[50].time := 3600.0, [116].log_data[50].minminute := 6, [116].log_data[50].maxminute := 15, [116].log_data[50].valid := 1, [116].log_data[51].time := 3600.0, [116].log_data[51].valid := 1, [116].log_data[52].min := -2.9199982, [116].log_data[52].max := 0.11999512, [116].log_data[52].total := -7780.122, [116].log_data[52].time := 3600.0, [116].log_data[52].minminute := 14, [116].log_data[52].maxminute := 2, [116].log_data[52].valid := 1, [116].log_data[53].min := -2.5600052, [116].log_data[53].max := 0.22000122, [116].log_data[53].total := -7581.878, [116].log_data[53].time := 3600.0, [116].log_data[53].minminute := 31, [116].log_data[53].maxminute := 19, [116].log_data[53].valid := 1,
        [116].log_data[54].max := 0.5265, [116].log_data[54].total := 1217.669, [116].log_data[54].time := 3600.0, [116].log_data[54].minminute := 2, [116].log_data[54].maxminute := 45, [116].log_data[54].valid := 1, [116].log_data[55].max := 0.52349997, [116].log_data[55].total := 1254.2191, [116].log_data[55].time := 3600.0, [116].log_data[55].minminute := 7, [116].log_data[55].maxminute := 30, [116].log_data[55].valid := 1, [116].log_data[56].min := 0.15934268, [116].log_data[56].max := 0.15981378, [116].log_data[56].total := 574.35345, [116].log_data[56].time := 3600.0, [116].log_data[56].minminute := 27, [116].log_data[56].maxminute := 37, [116].log_data[56].valid := 1, [116].log_data[57].min := 0.21622793, [116].log_data[57].max := 0.21846563, [116].log_data[57].total := 783.4741, [116].log_data[57].time := 3600.0, [116].log_data[57].minminute := 47, [116].log_data[57].maxminute := 28, [116].log_data[57].valid := 1, [116].log_data[58].time := 3600.0, [116].log_data[58].valid := 1, [116].log_data[59].time := 3600.0, [116].log_data[59].valid := 1, [116].log_data[60].valid := 1, [116].log_data[61].valid := 1, [116].log_data[62].valid := 1, [116].log_data[63].valid := 1, [116].log_data[64].valid := 1, [116].log_data[65].valid := 1, [116].log_data[66].valid := 1, [116].log_data[67].valid := 1, [116].log_data[68].valid := 1, [116].log_data[69].valid := 1, [116].log_data[70].valid := 1, [116].log_data[71].valid := 1, [116].log_data[72].valid := 1, [116].log_data[73].valid := 1, [116].log_data[74].valid := 1, [116].log_data[75].valid := 1, [116].log_data[76].valid := 1, [116].log_data[77].valid := 1, [116].log_data[78].valid := 1, [116].log_data[79].valid := 1, [116].log_data[80].valid := 1, [116].log_data[81].valid := 1, [116].log_data[82].valid := 1, [116].log_data[83].valid := 1, [116].log_data[84].valid := 1, [116].log_data[85].valid := 1, [116].log_data[86].valid := 1, [116].log_data[87].valid := 1, [116].log_data[88].valid := 1, [116].log_data[89].valid := 1,
        [116].log_data[90].valid := 1, [116].log_data[91].valid := 1, [116].log_data[92].valid := 1, [116].log_data[93].valid := 1, [116].log_data[94].valid := 1, [116].log_data[95].valid := 1, [116].log_data[96].valid := 1, [116].log_data[97].valid := 1, [116].log_data[98].valid := 1, [116].log_data[99].valid := 1, [116].log_data[100].valid := 1, [116].log_data[101].valid := 1, [116].log_data[102].valid := 1, [116].log_data[103].valid := 1, [116].log_data[104].valid := 1, [116].log_data[105].valid := 1, [116].log_data[106].valid := 1, [116].log_data[107].valid := 1, [116].log_data[108].valid := 1, [116].log_data[109].valid := 1, [116].log_data[110].valid := 1, [116].log_data[111].valid := 1, [116].log_data[112].valid := 1, [116].log_data[113].valid := 1, [116].log_data[114].valid := 1, [116].log_data[115].valid := 1, [116].log_data[116].valid := 1, [116].log_data[117].valid := 1, [116].log_data[118].valid := 1, [116].log_data[119].valid := 1, [116].log_data[120].valid := 1, [116].log_data[121].valid := 1, [116].log_data[122].valid := 1, [116].log_data[123].valid := 1, [116].log_data[124].valid := 1, [116].time.Year := 2023, [116].time.Month := 1, [116].time.Day := 17, [116].time.Hour := 23, [116].time.Minute := 59, [116].time.Second := 59, [117].log_data[0].min := 1.0, [117].log_data[0].max := 1.0, [117].log_data[0].total := 3600.0, [117].log_data[0].time := 3600.0, [117].log_data[0].valid := 1, [117].log_data[1].time := 3600.0, [117].log_data[1].valid := 1, [117].log_data[2].time := 3600.0, [117].log_data[2].valid := 1, [117].log_data[3].time := 3600.0, [117].log_data[3].valid := 1, [117].log_data[4].time := 3600.0, [117].log_data[4].valid := 1, [117].log_data[5].time := 3600.0, [117].log_data[5].valid := 1, [117].log_data[6].time := 3600.0, [117].log_data[6].valid := 1, [117].log_data[7].time := 3600.0, [117].log_data[7].valid := 1,
        [117].log_data[8].min := 1.0, [117].log_data[8].max := 1.0, [117].log_data[8].total := 3600.0, [117].log_data[8].time := 3600.0, [117].log_data[8].valid := 1, [117].log_data[9].min := 1.0, [117].log_data[9].max := 1.0, [117].log_data[9].total := 3600.0, [117].log_data[9].time := 3600.0, [117].log_data[9].valid := 1, [117].log_data[10].min := 1.0, [117].log_data[10].max := 1.0, [117].log_data[10].total := 3600.0, [117].log_data[10].time := 3600.0, [117].log_data[10].valid := 1, [117].log_data[11].time := 3600.0, [117].log_data[11].valid := 1, [117].log_data[12].min := 1.0, [117].log_data[12].max := 1.0, [117].log_data[12].total := 3600.0, [117].log_data[12].time := 3600.0, [117].log_data[12].valid := 1, [117].log_data[13].min := 1.0, [117].log_data[13].max := 1.0, [117].log_data[13].total := 3600.0, [117].log_data[13].time := 3600.0, [117].log_data[13].valid := 1, [117].log_data[14].time := 3600.0, [117].log_data[14].valid := 1, [117].log_data[15].time := 3600.0, [117].log_data[15].valid := 1, [117].log_data[16].time := 3600.0, [117].log_data[16].valid := 1, [117].log_data[17].min := 1.0, [117].log_data[17].max := 1.0, [117].log_data[17].total := 3600.0, [117].log_data[17].time := 3600.0, [117].log_data[17].valid := 1, [117].log_data[18].time := 3600.0, [117].log_data[18].valid := 1, [117].log_data[19].time := 3600.0, [117].log_data[19].valid := 1, [117].log_data[20].time := 3600.0, [117].log_data[20].valid := 1, [117].log_data[21].min := 1.0, [117].log_data[21].max := 1.0, [117].log_data[21].total := 3600.0, [117].log_data[21].time := 3600.0, [117].log_data[21].valid := 1, [117].log_data[22].time := 3600.0, [117].log_data[22].valid := 1, [117].log_data[23].time := 3600.0, [117].log_data[23].valid := 1, [117].log_data[24].time := 3600.0, [117].log_data[24].valid := 1, [117].log_data[25].time := 3600.0, [117].log_data[25].valid := 1, [117].log_data[26].time := 3600.0, [117].log_data[26].valid := 1, [117].log_data[27].time := 3600.0,
        [117].log_data[27].valid := 1, [117].log_data[28].time := 3600.0, [117].log_data[28].valid := 1, [117].log_data[29].min := 1.0, [117].log_data[29].max := 1.0, [117].log_data[29].total := 3600.0, [117].log_data[29].time := 3600.0, [117].log_data[29].valid := 1, [117].log_data[30].min := 1.0, [117].log_data[30].max := 1.0, [117].log_data[30].total := 3600.0, [117].log_data[30].time := 3600.0, [117].log_data[30].valid := 1, [117].log_data[31].max := 1.0, [117].log_data[31].total := 1440.998, [117].log_data[31].time := 3600.0, [117].log_data[31].minminute := 5, [117].log_data[31].valid := 1, [117].log_data[32].max := 1.0, [117].log_data[32].total := 1629.7471, [117].log_data[32].time := 3600.0, [117].log_data[32].maxminute := 6, [117].log_data[32].valid := 1, [117].log_data[33].time := 3600.0, [117].log_data[33].valid := 1, [117].log_data[34].time := 3600.0, [117].log_data[34].valid := 1, [117].log_data[35].max := 1.0, [117].log_data[35].total := 1440.7471, [117].log_data[35].time := 3600.0, [117].log_data[35].valid := 1, [117].log_data[36].max := 1.0, [117].log_data[36].total := 1629.7471, [117].log_data[36].time := 3600.0, [117].log_data[36].maxminute := 1, [117].log_data[36].valid := 1, [117].log_data[37].time := 3600.0, [117].log_data[37].valid := 1, [117].log_data[38].time := 3600.0, [117].log_data[38].valid := 1, [117].log_data[39].min := 0.9941174, [117].log_data[39].max := 1.0049527, [117].log_data[39].total := 3599.4175, [117].log_data[39].time := 3600.0, [117].log_data[39].minminute := 54, [117].log_data[39].maxminute := 12, [117].log_data[39].valid := 1, [117].log_data[40].min := 7.5816298, [117].log_data[40].max := 7.622027, [117].log_data[40].total := 27373.5, [117].log_data[40].time := 3600.0, [117].log_data[40].minminute := 30, [117].log_data[40].maxminute := 47, [117].log_data[40].valid := 1, [117].log_data[41].min := 0.02273633, [117].log_data[41].max := 0.023128908, [117].log_data[41].total := 82.58225, [117].log_data[41].time := 3600.0, [117].log_data[41].valid := 1, [117].log_data[42].min := 2.2917604,
        [117].log_data[42].max := 2.296118, [117].log_data[42].total := 8259.02, [117].log_data[42].time := 3600.0, [117].log_data[42].minminute := 55, [117].log_data[42].valid := 1, [117].log_data[43].min := -0.27999878, [117].log_data[43].max := -0.26000214, [117].log_data[43].total := -953.86755, [117].log_data[43].time := 3600.0, [117].log_data[43].valid := 1, [117].log_data[44].min := -0.3199997, [117].log_data[44].max := -0.30000305, [117].log_data[44].total := -1080.0961, [117].log_data[44].time := 3600.0, [117].log_data[44].minminute := 55, [117].log_data[44].valid := 1, [117].log_data[45].time := 3600.0, [117].log_data[45].valid := 1, [117].log_data[46].time := 3600.0, [117].log_data[46].valid := 1, [117].log_data[47].time := 3600.0, [117].log_data[47].valid := 1, [117].log_data[48].min := 6.7635264, [117].log_data[48].max := 6.792656, [117].log_data[48].total := 24376.98, [117].log_data[48].time := 3600.0, [117].log_data[48].minminute := 54, [117].log_data[48].valid := 1, [117].log_data[49].min := 8.882937, [117].log_data[49].max := 9.375824, [117].log_data[49].total := 33430.492, [117].log_data[49].time := 3600.0, [117].log_data[49].maxminute := 59, [117].log_data[49].valid := 1, [117].log_data[50].min := 1.8681242, [117].log_data[50].max := 1.9561024, [117].log_data[50].total := 6885.003, [117].log_data[50].time := 3600.0, [117].log_data[50].minminute := 59, [117].log_data[50].valid := 1, [117].log_data[51].time := 3600.0, [117].log_data[51].valid := 1, [117].log_data[52].min := -2.880005, [117].log_data[52].max := 0.11999512, [117].log_data[52].total := -7779.123, [117].log_data[52].time := 3600.0, [117].log_data[52].minminute := 27, [117].log_data[52].maxminute := 5, [117].log_data[52].valid := 1, [117].log_data[53].min := -2.7000046, [117].log_data[53].max := 0.27999878, [117].log_data[53].total := -7337.049, [117].log_data[53].time := 3600.0, [117].log_data[53].minminute := 12, [117].log_data[53].maxminute := 43, [117].log_data[53].valid := 1, [117].log_data[54].max := 0.541, [117].log_data[54].total := 1217.6157, [117].log_data[54].time := 3600.0, [117].log_data[54].minminute := 5,
        [117].log_data[54].maxminute := 38, [117].log_data[54].valid := 1, [117].log_data[55].max := 0.524, [117].log_data[55].total := 1217.3257, [117].log_data[55].time := 3600.0, [117].log_data[55].maxminute := 12, [117].log_data[55].valid := 1, [117].log_data[56].min := 0.15930341, [117].log_data[56].max := 0.15977451, [117].log_data[56].total := 574.32526, [117].log_data[56].time := 3600.0, [117].log_data[56].minminute := 53, [117].log_data[56].maxminute := 5, [117].log_data[56].valid := 1, [117].log_data[57].min := 0.21618867, [117].log_data[57].max := 0.21665977, [117].log_data[57].total := 779.1327, [117].log_data[57].time := 3600.0, [117].log_data[57].minminute := 31, [117].log_data[57].maxminute := 3, [117].log_data[57].valid := 1, [117].log_data[58].time := 3600.0, [117].log_data[58].valid := 1, [117].log_data[59].time := 3600.0, [117].log_data[59].valid := 1, [117].log_data[60].valid := 1, [117].log_data[61].valid := 1, [117].log_data[62].valid := 1, [117].log_data[63].valid := 1, [117].log_data[64].valid := 1, [117].log_data[65].valid := 1, [117].log_data[66].valid := 1, [117].log_data[67].valid := 1, [117].log_data[68].valid := 1, [117].log_data[69].valid := 1, [117].log_data[70].valid := 1, [117].log_data[71].valid := 1, [117].log_data[72].valid := 1, [117].log_data[73].valid := 1, [117].log_data[74].valid := 1, [117].log_data[75].valid := 1, [117].log_data[76].valid := 1, [117].log_data[77].valid := 1, [117].log_data[78].valid := 1, [117].log_data[79].valid := 1, [117].log_data[80].valid := 1, [117].log_data[81].valid := 1, [117].log_data[82].valid := 1, [117].log_data[83].valid := 1, [117].log_data[84].valid := 1, [117].log_data[85].valid := 1, [117].log_data[86].valid := 1, [117].log_data[87].valid := 1, [117].log_data[88].valid := 1, [117].log_data[89].valid := 1, [117].log_data[90].valid := 1, [117].log_data[91].valid := 1, [117].log_data[92].valid := 1, [117].log_data[93].valid := 1, [117].log_data[94].valid := 1,
        [117].log_data[95].valid := 1, [117].log_data[96].valid := 1, [117].log_data[97].valid := 1, [117].log_data[98].valid := 1, [117].log_data[99].valid := 1, [117].log_data[100].valid := 1, [117].log_data[101].valid := 1, [117].log_data[102].valid := 1, [117].log_data[103].valid := 1, [117].log_data[104].valid := 1, [117].log_data[105].valid := 1, [117].log_data[106].valid := 1, [117].log_data[107].valid := 1, [117].log_data[108].valid := 1, [117].log_data[109].valid := 1, [117].log_data[110].valid := 1, [117].log_data[111].valid := 1, [117].log_data[112].valid := 1, [117].log_data[113].valid := 1, [117].log_data[114].valid := 1, [117].log_data[115].valid := 1, [117].log_data[116].valid := 1, [117].log_data[117].valid := 1, [117].log_data[118].valid := 1, [117].log_data[119].valid := 1, [117].log_data[120].valid := 1, [117].log_data[121].valid := 1, [117].log_data[122].valid := 1, [117].log_data[123].valid := 1, [117].log_data[124].valid := 1, [117].time.Year := 2023, [117].time.Month := 1, [117].time.Day := 18, [117].time.Minute := 59, [117].time.Second := 59, [118].log_data[0].min := 1.0, [118].log_data[0].max := 1.0, [118].log_data[0].total := 3600.0, [118].log_data[0].time := 3600.0, [118].log_data[0].valid := 1, [118].log_data[1].max := 1.0, [118].log_data[1].total := 532.5, [118].log_data[1].time := 3600.0, [118].log_data[1].maxminute := 13, [118].log_data[1].valid := 1, [118].log_data[2].max := 1.0, [118].log_data[2].total := 529.0, [118].log_data[2].time := 3600.0, [118].log_data[2].maxminute := 13, [118].log_data[2].valid := 1, [118].log_data[3].time := 3600.0, [118].log_data[3].valid := 1, [118].log_data[4].time := 3600.0, [118].log_data[4].valid := 1, [118].log_data[5].max := 1.0, [118].log_data[5].total := 226.5, [118].log_data[5].time := 3600.0, [118].log_data[5].maxminute := 16, [118].log_data[5].valid := 1, [118].log_data[6].time := 3600.0,
        [118].log_data[6].valid := 1, [118].log_data[7].time := 3600.0, [118].log_data[7].valid := 1, [118].log_data[8].min := 1.0, [118].log_data[8].max := 1.0, [118].log_data[8].total := 3600.0, [118].log_data[8].time := 3600.0, [118].log_data[8].valid := 1, [118].log_data[9].min := 1.0, [118].log_data[9].max := 1.0, [118].log_data[9].total := 3600.0, [118].log_data[9].time := 3600.0, [118].log_data[9].valid := 1, [118].log_data[10].min := 1.0, [118].log_data[10].max := 1.0, [118].log_data[10].total := 3600.0, [118].log_data[10].time := 3600.0, [118].log_data[10].valid := 1, [118].log_data[11].time := 3600.0, [118].log_data[11].valid := 1, [118].log_data[12].min := 1.0, [118].log_data[12].max := 1.0, [118].log_data[12].total := 3600.0, [118].log_data[12].time := 3600.0, [118].log_data[12].valid := 1, [118].log_data[13].min := 1.0, [118].log_data[13].max := 1.0, [118].log_data[13].total := 3600.0, [118].log_data[13].time := 3600.0, [118].log_data[13].valid := 1, [118].log_data[14].time := 3600.0, [118].log_data[14].valid := 1, [118].log_data[15].time := 3600.0, [118].log_data[15].valid := 1, [118].log_data[16].time := 3600.0, [118].log_data[16].valid := 1, [118].log_data[17].min := 1.0, [118].log_data[17].max := 1.0, [118].log_data[17].total := 3600.0, [118].log_data[17].time := 3600.0, [118].log_data[17].valid := 1, [118].log_data[18].time := 3600.0, [118].log_data[18].valid := 1, [118].log_data[19].time := 3600.0, [118].log_data[19].valid := 1, [118].log_data[20].time := 3600.0, [118].log_data[20].valid := 1, [118].log_data[21].min := 1.0, [118].log_data[21].max := 1.0, [118].log_data[21].total := 3600.0, [118].log_data[21].time := 3600.0, [118].log_data[21].valid := 1, [118].log_data[22].time := 3600.0, [118].log_data[22].valid := 1, [118].log_data[23].time := 3600.0, [118].log_data[23].valid := 1, [118].log_data[24].time := 3600.0, [118].log_data[24].valid := 1, [118].log_data[25].time := 3600.0, [118].log_data[25].valid := 1,
        [118].log_data[26].time := 3600.0, [118].log_data[26].valid := 1, [118].log_data[27].time := 3600.0, [118].log_data[27].valid := 1, [118].log_data[28].time := 3600.0, [118].log_data[28].valid := 1, [118].log_data[29].min := 1.0, [118].log_data[29].max := 1.0, [118].log_data[29].total := 3600.0, [118].log_data[29].time := 3600.0, [118].log_data[29].valid := 1, [118].log_data[30].min := 1.0, [118].log_data[30].max := 1.0, [118].log_data[30].total := 3600.0, [118].log_data[30].time := 3600.0, [118].log_data[30].valid := 1, [118].log_data[31].max := 1.0, [118].log_data[31].total := 1591.249, [118].log_data[31].time := 3600.0, [118].log_data[31].minminute := 8, [118].log_data[31].valid := 1, [118].log_data[32].max := 1.0, [118].log_data[32].total := 1567.749, [118].log_data[32].time := 3600.0, [118].log_data[32].maxminute := 9, [118].log_data[32].valid := 1, [118].log_data[33].time := 3600.0, [118].log_data[33].valid := 1, [118].log_data[34].time := 3600.0, [118].log_data[34].valid := 1, [118].log_data[35].max := 1.0, [118].log_data[35].total := 1440.7471, [118].log_data[35].time := 3600.0, [118].log_data[35].minminute := 3, [118].log_data[35].valid := 1, [118].log_data[36].max := 1.0, [118].log_data[36].total := 1629.498, [118].log_data[36].time := 3600.0, [118].log_data[36].maxminute := 4, [118].log_data[36].valid := 1, [118].log_data[37].max := 7.5167155, [118].log_data[37].total := 3456.7234, [118].log_data[37].time := 3600.0, [118].log_data[37].maxminute := 15, [118].log_data[37].valid := 1, [118].log_data[38].time := 3600.0, [118].log_data[38].valid := 1, [118].log_data[39].min := 0.99423516, [118].log_data[39].max := 1.0217944, [118].log_data[39].total := 3606.87, [118].log_data[39].time := 3600.0, [118].log_data[39].minminute := 11, [118].log_data[39].maxminute := 16, [118].log_data[39].valid := 1, [118].log_data[40].min := 7.5959196, [118].log_data[40].max := 7.6179047, [118].log_data[40].total := 27381.592, [118].log_data[40].time := 3600.0, [118].log_data[40].minminute := 44, [118].log_data[40].valid := 1,
        [118].log_data[41].min := 0.02273633, [118].log_data[41].max := 0.023325196, [118].log_data[41].total := 82.57655, [118].log_data[41].time := 3600.0, [118].log_data[41].maxminute := 18, [118].log_data[41].valid := 1, [118].log_data[42].min := 2.291525, [118].log_data[42].max := 2.296236, [118].log_data[42].total := 8258.989, [118].log_data[42].time := 3600.0, [118].log_data[42].minminute := 49, [118].log_data[42].maxminute := 13, [118].log_data[42].valid := 1, [118].log_data[43].min := -0.27999878, [118].log_data[43].max := -0.26000214, [118].log_data[43].total := -950.2972, [118].log_data[43].time := 3600.0, [118].log_data[43].valid := 1, [118].log_data[44].min := -0.30000305, [118].log_data[44].max := -0.30000305, [118].log_data[44].total := -1080.0911, [118].log_data[44].time := 3600.0, [118].log_data[44].valid := 1, [118].log_data[45].time := 3600.0, [118].log_data[45].valid := 1, [118].log_data[46].time := 3600.0, [118].log_data[46].valid := 1, [118].log_data[47].time := 3600.0, [118].log_data[47].valid := 1, [118].log_data[48].min := 6.57968, [118].log_data[48].max := 6.9152203, [118].log_data[48].total := 24219.227, [118].log_data[48].time := 3600.0, [118].log_data[48].minminute := 45, [118].log_data[48].maxminute := 23, [118].log_data[48].valid := 1, [118].log_data[49].min := 6.6306896, [118].log_data[49].max := 9.39192, [118].log_data[49].total := 28958.957, [118].log_data[49].time := 3600.0, [118].log_data[49].minminute := 41, [118].log_data[49].maxminute := 15, [118].log_data[49].valid := 1, [118].log_data[50].min := 1.8451583, [118].log_data[50].max := 1.9450312, [118].log_data[50].total := 6852.9224, [118].log_data[50].time := 3600.0, [118].log_data[50].minminute := 16, [118].log_data[50].maxminute := 24, [118].log_data[50].valid := 1, [118].log_data[51].time := 3600.0, [118].log_data[51].valid := 1, [118].log_data[52].min := -3.0999985, [118].log_data[52].max := 0.11999512, [118].log_data[52].total := -8062.872, [118].log_data[52].time := 3600.0, [118].log_data[52].minminute := 20, [118].log_data[52].maxminute := 8, [118].log_data[52].valid := 1, [118].log_data[53].min := -2.6600037,
        [118].log_data[53].max := 0.19999695, [118].log_data[53].total := -7358.114, [118].log_data[53].time := 3600.0, [118].log_data[53].minminute := 36, [118].log_data[53].maxminute := 36, [118].log_data[53].valid := 1, [118].log_data[54].max := 0.5705, [118].log_data[54].total := 1254.5383, [118].log_data[54].time := 3600.0, [118].log_data[54].minminute := 8, [118].log_data[54].maxminute := 20, [118].log_data[54].valid := 1, [118].log_data[55].max := 0.5215, [118].log_data[55].total := 1217.1431, [118].log_data[55].time := 3600.0, [118].log_data[55].minminute := 3, [118].log_data[55].maxminute := 47, [118].log_data[55].valid := 1, [118].log_data[56].min := 0.15926416, [118].log_data[56].max := 0.15981378, [118].log_data[56].total := 574.288, [118].log_data[56].time := 3600.0, [118].log_data[56].minminute := 23, [118].log_data[56].maxminute := 3, [118].log_data[56].valid := 1, [118].log_data[57].min := 0.21438277, [118].log_data[57].max := 0.21673828, [118].log_data[57].total := 777.73315, [118].log_data[57].time := 3600.0, [118].log_data[57].minminute := 53, [118].log_data[57].valid := 1, [118].log_data[58].time := 3600.0, [118].log_data[58].valid := 1, [118].log_data[59].time := 3600.0, [118].log_data[59].valid := 1, [118].log_data[60].valid := 1, [118].log_data[61].valid := 1, [118].log_data[62].valid := 1, [118].log_data[63].valid := 1, [118].log_data[64].valid := 1, [118].log_data[65].valid := 1, [118].log_data[66].valid := 1, [118].log_data[67].valid := 1, [118].log_data[68].valid := 1, [118].log_data[69].valid := 1, [118].log_data[70].valid := 1, [118].log_data[71].valid := 1, [118].log_data[72].valid := 1, [118].log_data[73].valid := 1, [118].log_data[74].valid := 1, [118].log_data[75].valid := 1, [118].log_data[76].valid := 1, [118].log_data[77].valid := 1, [118].log_data[78].valid := 1, [118].log_data[79].valid := 1, [118].log_data[80].valid := 1, [118].log_data[81].valid := 1, [118].log_data[82].valid := 1, [118].log_data[83].valid := 1, [118].log_data[84].valid := 1,
        [118].log_data[85].valid := 1, [118].log_data[86].valid := 1, [118].log_data[87].valid := 1, [118].log_data[88].valid := 1, [118].log_data[89].valid := 1, [118].log_data[90].valid := 1, [118].log_data[91].valid := 1, [118].log_data[92].valid := 1, [118].log_data[93].valid := 1, [118].log_data[94].valid := 1, [118].log_data[95].valid := 1, [118].log_data[96].valid := 1, [118].log_data[97].valid := 1, [118].log_data[98].valid := 1, [118].log_data[99].valid := 1, [118].log_data[100].valid := 1, [118].log_data[101].valid := 1, [118].log_data[102].valid := 1, [118].log_data[103].valid := 1, [118].log_data[104].valid := 1, [118].log_data[105].valid := 1, [118].log_data[106].valid := 1, [118].log_data[107].valid := 1, [118].log_data[108].valid := 1, [118].log_data[109].valid := 1, [118].log_data[110].valid := 1, [118].log_data[111].valid := 1, [118].log_data[112].valid := 1, [118].log_data[113].valid := 1, [118].log_data[114].valid := 1, [118].log_data[115].valid := 1, [118].log_data[116].valid := 1, [118].log_data[117].valid := 1, [118].log_data[118].valid := 1, [118].log_data[119].valid := 1, [118].log_data[120].valid := 1, [118].log_data[121].valid := 1, [118].log_data[122].valid := 1, [118].log_data[123].valid := 1, [118].log_data[124].valid := 1, [118].time.Year := 2023, [118].time.Month := 1, [118].time.Day := 18, [118].time.Hour := 1, [118].time.Minute := 59, [118].time.Second := 59, [119].log_data[0].min := 1.0, [119].log_data[0].max := 1.0, [119].log_data[0].total := 3600.0, [119].log_data[0].time := 3600.0, [119].log_data[0].valid := 1, [119].log_data[1].time := 3600.0, [119].log_data[1].valid := 1, [119].log_data[2].time := 3600.0, [119].log_data[2].valid := 1, [119].log_data[3].time := 3600.0, [119].log_data[3].valid := 1, [119].log_data[4].time := 3600.0, [119].log_data[4].valid := 1, [119].log_data[5].time := 3600.0,
        [119].log_data[5].valid := 1, [119].log_data[6].time := 3600.0, [119].log_data[6].valid := 1, [119].log_data[7].time := 3600.0, [119].log_data[7].valid := 1, [119].log_data[8].min := 1.0, [119].log_data[8].max := 1.0, [119].log_data[8].total := 3600.0, [119].log_data[8].time := 3600.0, [119].log_data[8].valid := 1, [119].log_data[9].min := 1.0, [119].log_data[9].max := 1.0, [119].log_data[9].total := 3600.0, [119].log_data[9].time := 3600.0, [119].log_data[9].valid := 1, [119].log_data[10].min := 1.0, [119].log_data[10].max := 1.0, [119].log_data[10].total := 3600.0, [119].log_data[10].time := 3600.0, [119].log_data[10].valid := 1, [119].log_data[11].time := 3600.0, [119].log_data[11].valid := 1, [119].log_data[12].min := 1.0, [119].log_data[12].max := 1.0, [119].log_data[12].total := 3600.0, [119].log_data[12].time := 3600.0, [119].log_data[12].valid := 1, [119].log_data[13].min := 1.0, [119].log_data[13].max := 1.0, [119].log_data[13].total := 3600.0, [119].log_data[13].time := 3600.0, [119].log_data[13].valid := 1, [119].log_data[14].time := 3600.0, [119].log_data[14].valid := 1, [119].log_data[15].time := 3600.0, [119].log_data[15].valid := 1, [119].log_data[16].time := 3600.0, [119].log_data[16].valid := 1, [119].log_data[17].min := 1.0, [119].log_data[17].max := 1.0, [119].log_data[17].total := 3600.0, [119].log_data[17].time := 3600.0, [119].log_data[17].valid := 1, [119].log_data[18].time := 3600.0, [119].log_data[18].valid := 1, [119].log_data[19].time := 3600.0, [119].log_data[19].valid := 1, [119].log_data[20].time := 3600.0, [119].log_data[20].valid := 1, [119].log_data[21].min := 1.0, [119].log_data[21].max := 1.0, [119].log_data[21].total := 3600.0, [119].log_data[21].time := 3600.0, [119].log_data[21].valid := 1, [119].log_data[22].time := 3600.0, [119].log_data[22].valid := 1, [119].log_data[23].time := 3600.0, [119].log_data[23].valid := 1, [119].log_data[24].time := 3600.0, [119].log_data[24].valid := 1,
        [119].log_data[25].time := 3600.0, [119].log_data[25].valid := 1, [119].log_data[26].time := 3600.0, [119].log_data[26].valid := 1, [119].log_data[27].time := 3600.0, [119].log_data[27].valid := 1, [119].log_data[28].time := 3600.0, [119].log_data[28].valid := 1, [119].log_data[29].min := 1.0, [119].log_data[29].max := 1.0, [119].log_data[29].total := 3600.0, [119].log_data[29].time := 3600.0, [119].log_data[29].valid := 1, [119].log_data[30].min := 1.0, [119].log_data[30].max := 1.0, [119].log_data[30].total := 3600.0, [119].log_data[30].time := 3600.0, [119].log_data[30].valid := 1, [119].log_data[31].max := 1.0, [119].log_data[31].total := 1629.7471, [119].log_data[31].time := 3600.0, [119].log_data[31].maxminute := 2, [119].log_data[31].valid := 1, [119].log_data[32].max := 1.0, [119].log_data[32].total := 1440.998, [119].log_data[32].time := 3600.0, [119].log_data[32].minminute := 1, [119].log_data[32].valid := 1, [119].log_data[33].time := 3600.0, [119].log_data[33].valid := 1, [119].log_data[34].time := 3600.0, [119].log_data[34].valid := 1, [119].log_data[35].max := 1.0, [119].log_data[35].total := 1484.498, [119].log_data[35].time := 3600.0, [119].log_data[35].minminute := 6, [119].log_data[35].valid := 1, [119].log_data[36].max := 1.0, [119].log_data[36].total := 1629.998, [119].log_data[36].time := 3600.0, [119].log_data[36].maxminute := 8, [119].log_data[36].valid := 1, [119].log_data[37].time := 3600.0, [119].log_data[37].valid := 1, [119].log_data[38].time := 3600.0, [119].log_data[38].valid := 1, [119].log_data[39].min := 0.99541295, [119].log_data[39].max := 1.0050704, [119].log_data[39].total := 3603.2573, [119].log_data[39].time := 3600.0, [119].log_data[39].minminute := 54, [119].log_data[39].maxminute := 41, [119].log_data[39].valid := 1, [119].log_data[40].min := 7.6000414, [119].log_data[40].max := 7.6107597, [119].log_data[40].total := 27379.496, [119].log_data[40].time := 3600.0, [119].log_data[40].minminute := 15, [119].log_data[40].maxminute := 35, [119].log_data[40].valid := 1,
        [119].log_data[41].min := 0.02273633, [119].log_data[41].max := 0.023128908, [119].log_data[41].total := 82.56711, [119].log_data[41].time := 3600.0, [119].log_data[41].valid := 1, [119].log_data[42].min := 2.291525, [119].log_data[42].max := 2.2963536, [119].log_data[42].total := 8258.836, [119].log_data[42].time := 3600.0, [119].log_data[42].minminute := 15, [119].log_data[42].maxminute := 56, [119].log_data[42].valid := 1, [119].log_data[43].min := -0.27999878, [119].log_data[43].max := -0.26000214, [119].log_data[43].total := -950.7375, [119].log_data[43].time := 3600.0, [119].log_data[43].valid := 1, [119].log_data[44].min := -0.3199997, [119].log_data[44].max := -0.30000305, [119].log_data[44].total := -1080.0961, [119].log_data[44].time := 3600.0, [119].log_data[44].minminute := 20, [119].log_data[44].valid := 1, [119].log_data[45].time := 3600.0, [119].log_data[45].valid := 1, [119].log_data[46].time := 3600.0, [119].log_data[46].valid := 1, [119].log_data[47].time := 3600.0, [119].log_data[47].valid := 1, [119].log_data[48].min := 6.7489614, [119].log_data[48].max := 6.8041983, [119].log_data[48].total := 24355.51, [119].log_data[48].time := 3600.0, [119].log_data[48].minminute := 58, [119].log_data[48].valid := 1, [119].log_data[49].min := 8.507039, [119].log_data[49].max := 9.444135, [119].log_data[49].total := 33150.97, [119].log_data[49].time := 3600.0, [119].log_data[49].maxminute := 59, [119].log_data[49].valid := 1, [119].log_data[50].min := 1.8014638, [119].log_data[50].max := 1.9055767, [119].log_data[50].total := 6689.591, [119].log_data[50].time := 3600.0, [119].log_data[50].minminute := 59, [119].log_data[50].valid := 1, [119].log_data[51].time := 3600.0, [119].log_data[51].valid := 1, [119].log_data[52].min := -2.880005, [119].log_data[52].max := 0.11999512, [119].log_data[52].total := -7835.202, [119].log_data[52].time := 3600.0, [119].log_data[52].minminute := 23, [119].log_data[52].maxminute := 1, [119].log_data[52].valid := 1, [119].log_data[53].min := -2.6800003, [119].log_data[53].max := 0.19999695, [119].log_data[53].total := -7448.496, [119].log_data[53].time := 3600.0,
        [119].log_data[53].minminute := 18, [119].log_data[53].maxminute := 8, [119].log_data[53].valid := 1, [119].log_data[54].max := 0.515, [119].log_data[54].total := 1217.0316, [119].log_data[54].time := 3600.0, [119].log_data[54].minminute := 1, [119].log_data[54].maxminute := 23, [119].log_data[54].valid := 1, [119].log_data[55].max := 0.5415, [119].log_data[55].total := 1237.0873, [119].log_data[55].time := 3600.0, [119].log_data[55].minminute := 6, [119].log_data[55].maxminute := 18, [119].log_data[55].valid := 1, [119].log_data[56].min := 0.15930341, [119].log_data[56].max := 0.15981378, [119].log_data[56].total := 574.3376, [119].log_data[56].time := 3600.0, [119].log_data[56].minminute := 36, [119].log_data[56].maxminute := 10, [119].log_data[56].valid := 1, [119].log_data[57].min := 0.21438277, [119].log_data[57].max := 0.21485385, [119].log_data[57].total := 772.5691, [119].log_data[57].time := 3600.0, [119].log_data[57].minminute := 2, [119].log_data[57].maxminute := 33, [119].log_data[57].valid := 1, [119].log_data[58].time := 3600.0, [119].log_data[58].valid := 1, [119].log_data[59].time := 3600.0, [119].log_data[59].valid := 1, [119].log_data[60].valid := 1, [119].log_data[61].valid := 1, [119].log_data[62].valid := 1, [119].log_data[63].valid := 1, [119].log_data[64].valid := 1, [119].log_data[65].valid := 1, [119].log_data[66].valid := 1, [119].log_data[67].valid := 1, [119].log_data[68].valid := 1, [119].log_data[69].valid := 1, [119].log_data[70].valid := 1, [119].log_data[71].valid := 1, [119].log_data[72].valid := 1, [119].log_data[73].valid := 1, [119].log_data[74].valid := 1, [119].log_data[75].valid := 1, [119].log_data[76].valid := 1, [119].log_data[77].valid := 1, [119].log_data[78].valid := 1, [119].log_data[79].valid := 1, [119].log_data[80].valid := 1, [119].log_data[81].valid := 1, [119].log_data[82].valid := 1, [119].log_data[83].valid := 1, [119].log_data[84].valid := 1, [119].log_data[85].valid := 1, [119].log_data[86].valid := 1,
        [119].log_data[87].valid := 1, [119].log_data[88].valid := 1, [119].log_data[89].valid := 1, [119].log_data[90].valid := 1, [119].log_data[91].valid := 1, [119].log_data[92].valid := 1, [119].log_data[93].valid := 1, [119].log_data[94].valid := 1, [119].log_data[95].valid := 1, [119].log_data[96].valid := 1, [119].log_data[97].valid := 1, [119].log_data[98].valid := 1, [119].log_data[99].valid := 1, [119].log_data[100].valid := 1, [119].log_data[101].valid := 1, [119].log_data[102].valid := 1, [119].log_data[103].valid := 1, [119].log_data[104].valid := 1, [119].log_data[105].valid := 1, [119].log_data[106].valid := 1, [119].log_data[107].valid := 1, [119].log_data[108].valid := 1, [119].log_data[109].valid := 1, [119].log_data[110].valid := 1, [119].log_data[111].valid := 1, [119].log_data[112].valid := 1, [119].log_data[113].valid := 1, [119].log_data[114].valid := 1, [119].log_data[115].valid := 1, [119].log_data[116].valid := 1, [119].log_data[117].valid := 1, [119].log_data[118].valid := 1, [119].log_data[119].valid := 1, [119].log_data[120].valid := 1, [119].log_data[121].valid := 1, [119].log_data[122].valid := 1, [119].log_data[123].valid := 1, [119].log_data[124].valid := 1, [119].time.Year := 2023, [119].time.Month := 1, [119].time.Day := 18, [119].time.Hour := 2, [119].time.Minute := 59, [119].time.Second := 59, [120].log_data[0].min := 1.0, [120].log_data[0].max := 1.0, [120].log_data[0].total := 3600.0, [120].log_data[0].time := 3600.0, [120].log_data[0].valid := 1, [120].log_data[1].time := 3600.0, [120].log_data[1].valid := 1, [120].log_data[2].time := 3600.0, [120].log_data[2].valid := 1, [120].log_data[3].time := 3600.0, [120].log_data[3].valid := 1, [120].log_data[4].time := 3600.0, [120].log_data[4].valid := 1, [120].log_data[5].time := 3600.0, [120].log_data[5].valid := 1, [120].log_data[6].time := 3600.0,
        [120].log_data[6].valid := 1, [120].log_data[7].time := 3600.0, [120].log_data[7].valid := 1, [120].log_data[8].min := 1.0, [120].log_data[8].max := 1.0, [120].log_data[8].total := 3600.0, [120].log_data[8].time := 3600.0, [120].log_data[8].valid := 1, [120].log_data[9].min := 1.0, [120].log_data[9].max := 1.0, [120].log_data[9].total := 3600.0, [120].log_data[9].time := 3600.0, [120].log_data[9].valid := 1, [120].log_data[10].min := 1.0, [120].log_data[10].max := 1.0, [120].log_data[10].total := 3600.0, [120].log_data[10].time := 3600.0, [120].log_data[10].valid := 1, [120].log_data[11].time := 3600.0, [120].log_data[11].valid := 1, [120].log_data[12].min := 1.0, [120].log_data[12].max := 1.0, [120].log_data[12].total := 3600.0, [120].log_data[12].time := 3600.0, [120].log_data[12].valid := 1, [120].log_data[13].min := 1.0, [120].log_data[13].max := 1.0, [120].log_data[13].total := 3600.0, [120].log_data[13].time := 3600.0, [120].log_data[13].valid := 1, [120].log_data[14].time := 3600.0, [120].log_data[14].valid := 1, [120].log_data[15].time := 3600.0, [120].log_data[15].valid := 1, [120].log_data[16].time := 3600.0, [120].log_data[16].valid := 1, [120].log_data[17].min := 1.0, [120].log_data[17].max := 1.0, [120].log_data[17].total := 3600.0, [120].log_data[17].time := 3600.0, [120].log_data[17].valid := 1, [120].log_data[18].time := 3600.0, [120].log_data[18].valid := 1, [120].log_data[19].time := 3600.0, [120].log_data[19].valid := 1, [120].log_data[20].time := 3600.0, [120].log_data[20].valid := 1, [120].log_data[21].min := 1.0, [120].log_data[21].max := 1.0, [120].log_data[21].total := 3600.0, [120].log_data[21].time := 3600.0, [120].log_data[21].valid := 1, [120].log_data[22].time := 3600.0, [120].log_data[22].valid := 1, [120].log_data[23].time := 3600.0, [120].log_data[23].valid := 1, [120].log_data[24].time := 3600.0, [120].log_data[24].valid := 1, [120].log_data[25].time := 3600.0, [120].log_data[25].valid := 1,
        [120].log_data[26].time := 3600.0, [120].log_data[26].valid := 1, [120].log_data[27].time := 3600.0, [120].log_data[27].valid := 1, [120].log_data[28].time := 3600.0, [120].log_data[28].valid := 1, [120].log_data[29].min := 1.0, [120].log_data[29].max := 1.0, [120].log_data[29].total := 3600.0, [120].log_data[29].time := 3600.0, [120].log_data[29].valid := 1, [120].log_data[30].min := 1.0, [120].log_data[30].max := 1.0, [120].log_data[30].total := 3600.0, [120].log_data[30].time := 3600.0, [120].log_data[30].valid := 1, [120].log_data[31].max := 1.0, [120].log_data[31].total := 1629.7471, [120].log_data[31].time := 3600.0, [120].log_data[31].maxminute := 5, [120].log_data[31].valid := 1, [120].log_data[32].max := 1.0, [120].log_data[32].total := 1440.7471, [120].log_data[32].time := 3600.0, [120].log_data[32].minminute := 4, [120].log_data[32].valid := 1, [120].log_data[33].time := 3600.0, [120].log_data[33].valid := 1, [120].log_data[34].time := 3600.0, [120].log_data[34].valid := 1, [120].log_data[35].max := 1.0, [120].log_data[35].total := 1629.7471, [120].log_data[35].time := 3600.0, [120].log_data[35].valid := 1, [120].log_data[36].max := 1.0, [120].log_data[36].total := 1485.2471, [120].log_data[36].time := 3600.0, [120].log_data[36].maxminute := 11, [120].log_data[36].valid := 1, [120].log_data[37].time := 3600.0, [120].log_data[37].valid := 1, [120].log_data[38].time := 3600.0, [120].log_data[38].valid := 1, [120].log_data[39].min := 0.9956484, [120].log_data[39].max := 1.0048349, [120].log_data[39].total := 3603.893, [120].log_data[39].time := 3600.0, [120].log_data[39].minminute := 40, [120].log_data[39].maxminute := 5, [120].log_data[39].valid := 1, [120].log_data[40].min := 7.581355, [120].log_data[40].max := 7.6206527, [120].log_data[40].total := 27379.639, [120].log_data[40].time := 3600.0, [120].log_data[40].minminute := 51, [120].log_data[40].maxminute := 55, [120].log_data[40].valid := 1, [120].log_data[41].min := 0.02273633, [120].log_data[41].max := 0.023128908, [120].log_data[41].total := 82.46608,
        [120].log_data[41].time := 3600.0, [120].log_data[41].valid := 1, [120].log_data[42].min := 2.2918782, [120].log_data[42].max := 2.296236, [120].log_data[42].total := 8258.726, [120].log_data[42].time := 3600.0, [120].log_data[42].minminute := 43, [120].log_data[42].maxminute := 13, [120].log_data[42].valid := 1, [120].log_data[43].min := -0.27999878, [120].log_data[43].max := -0.26000214, [120].log_data[43].total := -941.9987, [120].log_data[43].time := 3600.0, [120].log_data[43].valid := 1, [120].log_data[44].min := -0.30000305, [120].log_data[44].max := -0.30000305, [120].log_data[44].total := -1080.0911, [120].log_data[44].time := 3600.0, [120].log_data[44].valid := 1, [120].log_data[45].time := 3600.0, [120].log_data[45].valid := 1, [120].log_data[46].time := 3600.0, [120].log_data[46].valid := 1, [120].log_data[47].time := 3600.0, [120].log_data[47].valid := 1, [120].log_data[48].min := 6.729175, [120].log_data[48].max := 6.752809, [120].log_data[48].total := 24267.59, [120].log_data[48].time := 3600.0, [120].log_data[48].minminute := 57, [120].log_data[48].valid := 1, [120].log_data[49].min := 9.410175, [120].log_data[49].max := 9.600971, [120].log_data[49].total := 34220.203, [120].log_data[49].time := 3600.0, [120].log_data[49].maxminute := 19, [120].log_data[49].valid := 1, [120].log_data[50].min := 1.7269124, [120].log_data[50].max := 1.8112392, [120].log_data[50].total := 6365.1807, [120].log_data[50].time := 3600.0, [120].log_data[50].minminute := 59, [120].log_data[50].maxminute := 2, [120].log_data[50].valid := 1, [120].log_data[51].time := 3600.0, [120].log_data[51].valid := 1, [120].log_data[52].min := -2.880005, [120].log_data[52].max := 0.11999512, [120].log_data[52].total := -7831.628, [120].log_data[52].time := 3600.0, [120].log_data[52].minminute := 26, [120].log_data[52].maxminute := 4, [120].log_data[52].valid := 1, [120].log_data[53].min := -2.600006, [120].log_data[53].max := 0.22000122, [120].log_data[53].total := -7482.3647, [120].log_data[53].time := 3600.0, [120].log_data[53].minminute := 2, [120].log_data[53].maxminute := 10, [120].log_data[53].valid := 1,
        [120].log_data[54].max := 0.543, [120].log_data[54].total := 1217.3976, [120].log_data[54].time := 3600.0, [120].log_data[54].minminute := 4, [120].log_data[54].maxminute := 26, [120].log_data[54].valid := 1, [120].log_data[55].max := 0.532, [120].log_data[55].total := 1234.5597, [120].log_data[55].time := 3600.0, [120].log_data[55].valid := 1, [120].log_data[56].min := 0.15930341, [120].log_data[56].max := 0.15981378, [120].log_data[56].total := 574.2402, [120].log_data[56].time := 3600.0, [120].log_data[56].minminute := 7, [120].log_data[56].valid := 1, [120].log_data[57].min := 0.21450053, [120].log_data[57].max := 0.21493237, [120].log_data[57].total := 772.8753, [120].log_data[57].time := 3600.0, [120].log_data[57].minminute := 19, [120].log_data[57].maxminute := 26, [120].log_data[57].valid := 1, [120].log_data[58].time := 3600.0, [120].log_data[58].valid := 1, [120].log_data[59].time := 3600.0, [120].log_data[59].valid := 1, [120].log_data[60].valid := 1, [120].log_data[61].valid := 1, [120].log_data[62].valid := 1, [120].log_data[63].valid := 1, [120].log_data[64].valid := 1, [120].log_data[65].valid := 1, [120].log_data[66].valid := 1, [120].log_data[67].valid := 1, [120].log_data[68].valid := 1, [120].log_data[69].valid := 1, [120].log_data[70].valid := 1, [120].log_data[71].valid := 1, [120].log_data[72].valid := 1, [120].log_data[73].valid := 1, [120].log_data[74].valid := 1, [120].log_data[75].valid := 1, [120].log_data[76].valid := 1, [120].log_data[77].valid := 1, [120].log_data[78].valid := 1, [120].log_data[79].valid := 1, [120].log_data[80].valid := 1, [120].log_data[81].valid := 1, [120].log_data[82].valid := 1, [120].log_data[83].valid := 1, [120].log_data[84].valid := 1, [120].log_data[85].valid := 1, [120].log_data[86].valid := 1, [120].log_data[87].valid := 1, [120].log_data[88].valid := 1, [120].log_data[89].valid := 1, [120].log_data[90].valid := 1, [120].log_data[91].valid := 1, [120].log_data[92].valid := 1,
        [120].log_data[93].valid := 1, [120].log_data[94].valid := 1, [120].log_data[95].valid := 1, [120].log_data[96].valid := 1, [120].log_data[97].valid := 1, [120].log_data[98].valid := 1, [120].log_data[99].valid := 1, [120].log_data[100].valid := 1, [120].log_data[101].valid := 1, [120].log_data[102].valid := 1, [120].log_data[103].valid := 1, [120].log_data[104].valid := 1, [120].log_data[105].valid := 1, [120].log_data[106].valid := 1, [120].log_data[107].valid := 1, [120].log_data[108].valid := 1, [120].log_data[109].valid := 1, [120].log_data[110].valid := 1, [120].log_data[111].valid := 1, [120].log_data[112].valid := 1, [120].log_data[113].valid := 1, [120].log_data[114].valid := 1, [120].log_data[115].valid := 1, [120].log_data[116].valid := 1, [120].log_data[117].valid := 1, [120].log_data[118].valid := 1, [120].log_data[119].valid := 1, [120].log_data[120].valid := 1, [120].log_data[121].valid := 1, [120].log_data[122].valid := 1, [120].log_data[123].valid := 1, [120].log_data[124].valid := 1, [120].time.Year := 2023, [120].time.Month := 1, [120].time.Day := 18, [120].time.Hour := 3, [120].time.Minute := 59, [120].time.Second := 59, [121].log_data[0].min := 1.0, [121].log_data[0].max := 1.0, [121].log_data[0].total := 3600.0, [121].log_data[0].time := 3600.0, [121].log_data[0].valid := 1, [121].log_data[1].time := 3600.0, [121].log_data[1].valid := 1, [121].log_data[2].time := 3600.0, [121].log_data[2].valid := 1, [121].log_data[3].time := 3600.0, [121].log_data[3].valid := 1, [121].log_data[4].time := 3600.0, [121].log_data[4].valid := 1, [121].log_data[5].time := 3600.0, [121].log_data[5].valid := 1, [121].log_data[6].time := 3600.0, [121].log_data[6].valid := 1, [121].log_data[7].time := 3600.0, [121].log_data[7].valid := 1, [121].log_data[8].min := 1.0, [121].log_data[8].max := 1.0, [121].log_data[8].total := 3600.0,
        [121].log_data[8].time := 3600.0, [121].log_data[8].valid := 1, [121].log_data[9].min := 1.0, [121].log_data[9].max := 1.0, [121].log_data[9].total := 3600.0, [121].log_data[9].time := 3600.0, [121].log_data[9].valid := 1, [121].log_data[10].min := 1.0, [121].log_data[10].max := 1.0, [121].log_data[10].total := 3600.0, [121].log_data[10].time := 3600.0, [121].log_data[10].valid := 1, [121].log_data[11].time := 3600.0, [121].log_data[11].valid := 1, [121].log_data[12].min := 1.0, [121].log_data[12].max := 1.0, [121].log_data[12].total := 3600.0, [121].log_data[12].time := 3600.0, [121].log_data[12].valid := 1, [121].log_data[13].min := 1.0, [121].log_data[13].max := 1.0, [121].log_data[13].total := 3600.0, [121].log_data[13].time := 3600.0, [121].log_data[13].valid := 1, [121].log_data[14].time := 3600.0, [121].log_data[14].valid := 1, [121].log_data[15].time := 3600.0, [121].log_data[15].valid := 1, [121].log_data[16].time := 3600.0, [121].log_data[16].valid := 1, [121].log_data[17].min := 1.0, [121].log_data[17].max := 1.0, [121].log_data[17].total := 3600.0, [121].log_data[17].time := 3600.0, [121].log_data[17].valid := 1, [121].log_data[18].time := 3600.0, [121].log_data[18].valid := 1, [121].log_data[19].time := 3600.0, [121].log_data[19].valid := 1, [121].log_data[20].time := 3600.0, [121].log_data[20].valid := 1, [121].log_data[21].min := 1.0, [121].log_data[21].max := 1.0, [121].log_data[21].total := 3600.0, [121].log_data[21].time := 3600.0, [121].log_data[21].valid := 1, [121].log_data[22].time := 3600.0, [121].log_data[22].valid := 1, [121].log_data[23].time := 3600.0, [121].log_data[23].valid := 1, [121].log_data[24].time := 3600.0, [121].log_data[24].valid := 1, [121].log_data[25].time := 3600.0, [121].log_data[25].valid := 1, [121].log_data[26].time := 3600.0, [121].log_data[26].valid := 1, [121].log_data[27].time := 3600.0, [121].log_data[27].valid := 1, [121].log_data[28].time := 3600.0, [121].log_data[28].valid := 1,
        [121].log_data[29].min := 1.0, [121].log_data[29].max := 1.0, [121].log_data[29].total := 3600.0, [121].log_data[29].time := 3600.0, [121].log_data[29].valid := 1, [121].log_data[30].min := 1.0, [121].log_data[30].max := 1.0, [121].log_data[30].total := 3600.0, [121].log_data[30].time := 3600.0, [121].log_data[30].valid := 1, [121].log_data[31].max := 1.0, [121].log_data[31].total := 1629.7471, [121].log_data[31].time := 3600.0, [121].log_data[31].maxminute := 8, [121].log_data[31].valid := 1, [121].log_data[32].max := 1.0, [121].log_data[32].total := 1526.998, [121].log_data[32].time := 3600.0, [121].log_data[32].minminute := 7, [121].log_data[32].valid := 1, [121].log_data[33].time := 3600.0, [121].log_data[33].valid := 1, [121].log_data[34].time := 3600.0, [121].log_data[34].valid := 1, [121].log_data[35].max := 1.0, [121].log_data[35].total := 1629.7471, [121].log_data[35].time := 3600.0, [121].log_data[35].maxminute := 3, [121].log_data[35].valid := 1, [121].log_data[36].max := 1.0, [121].log_data[36].total := 1440.7471, [121].log_data[36].time := 3600.0, [121].log_data[36].minminute := 2, [121].log_data[36].valid := 1, [121].log_data[37].time := 3600.0, [121].log_data[37].valid := 1, [121].log_data[38].time := 3600.0, [121].log_data[38].valid := 1, [121].log_data[39].min := 0.9944707, [121].log_data[39].max := 1.0050704, [121].log_data[39].total := 3604.2861, [121].log_data[39].time := 3600.0, [121].log_data[39].minminute := 20, [121].log_data[39].maxminute := 3, [121].log_data[39].valid := 1, [121].log_data[40].min := 7.588774, [121].log_data[40].max := 7.6107597, [121].log_data[40].total := 27381.457, [121].log_data[40].time := 3600.0, [121].log_data[40].minminute := 8, [121].log_data[40].maxminute := 16, [121].log_data[40].valid := 1, [121].log_data[41].min := 0.022540038, [121].log_data[41].max := 0.023128908, [121].log_data[41].total := 82.33516, [121].log_data[41].time := 3600.0, [121].log_data[41].minminute := 4, [121].log_data[41].valid := 1, [121].log_data[42].min := 2.2907004, [121].log_data[42].max := 2.2965894,
        [121].log_data[42].total := 8258.586, [121].log_data[42].time := 3600.0, [121].log_data[42].minminute := 17, [121].log_data[42].maxminute := 31, [121].log_data[42].valid := 1, [121].log_data[43].min := -0.27999878, [121].log_data[43].max := -0.26000214, [121].log_data[43].total := -937.4094, [121].log_data[43].time := 3600.0, [121].log_data[43].valid := 1, [121].log_data[44].min := -0.30000305, [121].log_data[44].max := -0.30000305, [121].log_data[44].total := -1080.0911, [121].log_data[44].time := 3600.0, [121].log_data[44].valid := 1, [121].log_data[45].time := 3600.0, [121].log_data[45].valid := 1, [121].log_data[46].time := 3600.0, [121].log_data[46].valid := 1, [121].log_data[47].time := 3600.0, [121].log_data[47].valid := 1, [121].log_data[48].min := 6.694824, [121].log_data[48].max := 6.7299995, [121].log_data[48].total := 24168.688, [121].log_data[48].time := 3600.0, [121].log_data[48].minminute := 58, [121].log_data[48].maxminute := 4, [121].log_data[48].valid := 1, [121].log_data[49].min := 9.444722, [121].log_data[49].max := 9.516173, [121].log_data[49].total := 34137.05, [121].log_data[49].time := 3600.0, [121].log_data[49].minminute := 58, [121].log_data[49].maxminute := 21, [121].log_data[49].valid := 1, [121].log_data[50].min := 1.6308081, [121].log_data[50].max := 1.7317412, [121].log_data[50].total := 6069.012, [121].log_data[50].time := 3600.0, [121].log_data[50].minminute := 59, [121].log_data[50].valid := 1, [121].log_data[51].time := 3600.0, [121].log_data[51].valid := 1, [121].log_data[52].min := -2.8600006, [121].log_data[52].max := 0.11999512, [121].log_data[52].total := -8100.049, [121].log_data[52].time := 3600.0, [121].log_data[52].minminute := 50, [121].log_data[52].maxminute := 7, [121].log_data[52].valid := 1, [121].log_data[53].min := -2.6200027, [121].log_data[53].max := 0.13999939, [121].log_data[53].total := -7438.403, [121].log_data[53].time := 3600.0, [121].log_data[53].minminute := 32, [121].log_data[53].maxminute := 3, [121].log_data[53].valid := 1, [121].log_data[54].max := 0.513, [121].log_data[54].total := 1253.8058, [121].log_data[54].time := 3600.0,
        [121].log_data[54].minminute := 7, [121].log_data[54].maxminute := 40, [121].log_data[54].valid := 1, [121].log_data[55].max := 0.517, [121].log_data[55].total := 1217.0637, [121].log_data[55].time := 3600.0, [121].log_data[55].minminute := 2, [121].log_data[55].maxminute := 25, [121].log_data[55].valid := 1, [121].log_data[56].min := 0.15926416, [121].log_data[56].max := 0.15973525, [121].log_data[56].total := 574.0682, [121].log_data[56].time := 3600.0, [121].log_data[56].minminute := 5, [121].log_data[56].valid := 1, [121].log_data[57].min := 0.2145398, [121].log_data[57].max := 0.21497163, [121].log_data[57].total := 772.9762, [121].log_data[57].time := 3600.0, [121].log_data[57].maxminute := 46, [121].log_data[57].valid := 1, [121].log_data[58].time := 3600.0, [121].log_data[58].valid := 1, [121].log_data[59].time := 3600.0, [121].log_data[59].valid := 1, [121].log_data[60].valid := 1, [121].log_data[61].valid := 1, [121].log_data[62].valid := 1, [121].log_data[63].valid := 1, [121].log_data[64].valid := 1, [121].log_data[65].valid := 1, [121].log_data[66].valid := 1, [121].log_data[67].valid := 1, [121].log_data[68].valid := 1, [121].log_data[69].valid := 1, [121].log_data[70].valid := 1, [121].log_data[71].valid := 1, [121].log_data[72].valid := 1, [121].log_data[73].valid := 1, [121].log_data[74].valid := 1, [121].log_data[75].valid := 1, [121].log_data[76].valid := 1, [121].log_data[77].valid := 1, [121].log_data[78].valid := 1, [121].log_data[79].valid := 1, [121].log_data[80].valid := 1, [121].log_data[81].valid := 1, [121].log_data[82].valid := 1, [121].log_data[83].valid := 1, [121].log_data[84].valid := 1, [121].log_data[85].valid := 1, [121].log_data[86].valid := 1, [121].log_data[87].valid := 1, [121].log_data[88].valid := 1, [121].log_data[89].valid := 1, [121].log_data[90].valid := 1, [121].log_data[91].valid := 1, [121].log_data[92].valid := 1, [121].log_data[93].valid := 1, [121].log_data[94].valid := 1,
        [121].log_data[95].valid := 1, [121].log_data[96].valid := 1, [121].log_data[97].valid := 1, [121].log_data[98].valid := 1, [121].log_data[99].valid := 1, [121].log_data[100].valid := 1, [121].log_data[101].valid := 1, [121].log_data[102].valid := 1, [121].log_data[103].valid := 1, [121].log_data[104].valid := 1, [121].log_data[105].valid := 1, [121].log_data[106].valid := 1, [121].log_data[107].valid := 1, [121].log_data[108].valid := 1, [121].log_data[109].valid := 1, [121].log_data[110].valid := 1, [121].log_data[111].valid := 1, [121].log_data[112].valid := 1, [121].log_data[113].valid := 1, [121].log_data[114].valid := 1, [121].log_data[115].valid := 1, [121].log_data[116].valid := 1, [121].log_data[117].valid := 1, [121].log_data[118].valid := 1, [121].log_data[119].valid := 1, [121].log_data[120].valid := 1, [121].log_data[121].valid := 1, [121].log_data[122].valid := 1, [121].log_data[123].valid := 1, [121].log_data[124].valid := 1, [121].time.Year := 2023, [121].time.Month := 1, [121].time.Day := 18, [121].time.Hour := 4, [121].time.Minute := 59, [121].time.Second := 59, [122].log_data[0].min := 1.0, [122].log_data[0].max := 1.0, [122].log_data[0].total := 3600.0, [122].log_data[0].time := 3600.0, [122].log_data[0].valid := 1, [122].log_data[1].max := 1.0, [122].log_data[1].total := 532.0, [122].log_data[1].time := 3600.0, [122].log_data[1].maxminute := 27, [122].log_data[1].valid := 1, [122].log_data[2].max := 1.0, [122].log_data[2].total := 528.5, [122].log_data[2].time := 3600.0, [122].log_data[2].maxminute := 27, [122].log_data[2].valid := 1, [122].log_data[3].time := 3600.0, [122].log_data[3].valid := 1, [122].log_data[4].time := 3600.0, [122].log_data[4].valid := 1, [122].log_data[5].max := 1.0, [122].log_data[5].total := 224.5, [122].log_data[5].time := 3600.0, [122].log_data[5].maxminute := 30, [122].log_data[5].valid := 1,
        [122].log_data[6].time := 3600.0, [122].log_data[6].valid := 1, [122].log_data[7].time := 3600.0, [122].log_data[7].valid := 1, [122].log_data[8].min := 1.0, [122].log_data[8].max := 1.0, [122].log_data[8].total := 3600.0, [122].log_data[8].time := 3600.0, [122].log_data[8].valid := 1, [122].log_data[9].min := 1.0, [122].log_data[9].max := 1.0, [122].log_data[9].total := 3600.0, [122].log_data[9].time := 3600.0, [122].log_data[9].valid := 1, [122].log_data[10].min := 1.0, [122].log_data[10].max := 1.0, [122].log_data[10].total := 3600.0, [122].log_data[10].time := 3600.0, [122].log_data[10].valid := 1, [122].log_data[11].time := 3600.0, [122].log_data[11].valid := 1, [122].log_data[12].min := 1.0, [122].log_data[12].max := 1.0, [122].log_data[12].total := 3600.0, [122].log_data[12].time := 3600.0, [122].log_data[12].valid := 1, [122].log_data[13].min := 1.0, [122].log_data[13].max := 1.0, [122].log_data[13].total := 3600.0, [122].log_data[13].time := 3600.0, [122].log_data[13].valid := 1, [122].log_data[14].time := 3600.0, [122].log_data[14].valid := 1, [122].log_data[15].time := 3600.0, [122].log_data[15].valid := 1, [122].log_data[16].time := 3600.0, [122].log_data[16].valid := 1, [122].log_data[17].min := 1.0, [122].log_data[17].max := 1.0, [122].log_data[17].total := 3600.0, [122].log_data[17].time := 3600.0, [122].log_data[17].valid := 1, [122].log_data[18].time := 3600.0, [122].log_data[18].valid := 1, [122].log_data[19].time := 3600.0, [122].log_data[19].valid := 1, [122].log_data[20].time := 3600.0, [122].log_data[20].valid := 1, [122].log_data[21].min := 1.0, [122].log_data[21].max := 1.0, [122].log_data[21].total := 3600.0, [122].log_data[21].time := 3600.0, [122].log_data[21].valid := 1, [122].log_data[22].time := 3600.0, [122].log_data[22].valid := 1, [122].log_data[23].time := 3600.0, [122].log_data[23].valid := 1, [122].log_data[24].time := 3600.0, [122].log_data[24].valid := 1, [122].log_data[25].time := 3600.0,
        [122].log_data[25].valid := 1, [122].log_data[26].time := 3600.0, [122].log_data[26].valid := 1, [122].log_data[27].time := 3600.0, [122].log_data[27].valid := 1, [122].log_data[28].time := 3600.0, [122].log_data[28].valid := 1, [122].log_data[29].min := 1.0, [122].log_data[29].max := 1.0, [122].log_data[29].total := 3600.0, [122].log_data[29].time := 3600.0, [122].log_data[29].valid := 1, [122].log_data[30].min := 1.0, [122].log_data[30].max := 1.0, [122].log_data[30].total := 3600.0, [122].log_data[30].time := 3600.0, [122].log_data[30].valid := 1, [122].log_data[31].max := 1.0, [122].log_data[31].total := 1442.2471, [122].log_data[31].time := 3600.0, [122].log_data[31].maxminute := 11, [122].log_data[31].valid := 1, [122].log_data[32].max := 1.0, [122].log_data[32].total := 1629.998, [122].log_data[32].time := 3600.0, [122].log_data[32].maxminute := 1, [122].log_data[32].valid := 1, [122].log_data[33].time := 3600.0, [122].log_data[33].valid := 1, [122].log_data[34].time := 3600.0, [122].log_data[34].valid := 1, [122].log_data[35].max := 1.0, [122].log_data[35].total := 1629.998, [122].log_data[35].time := 3600.0, [122].log_data[35].maxminute := 7, [122].log_data[35].valid := 1, [122].log_data[36].max := 1.0, [122].log_data[36].total := 1440.2471, [122].log_data[36].time := 3600.0, [122].log_data[36].minminute := 5, [122].log_data[36].valid := 1, [122].log_data[37].max := 7.3698897, [122].log_data[37].total := 3383.3787, [122].log_data[37].time := 3600.0, [122].log_data[37].maxminute := 28, [122].log_data[37].valid := 1, [122].log_data[38].time := 3600.0, [122].log_data[38].valid := 1, [122].log_data[39].min := 0.9961195, [122].log_data[39].max := 1.0207345, [122].log_data[39].total := 3609.8647, [122].log_data[39].time := 3600.0, [122].log_data[39].minminute := 32, [122].log_data[39].maxminute := 30, [122].log_data[39].valid := 1, [122].log_data[40].min := 7.5970187, [122].log_data[40].max := 7.6135077, [122].log_data[40].total := 27382.383, [122].log_data[40].time := 3600.0, [122].log_data[40].minminute := 3,
